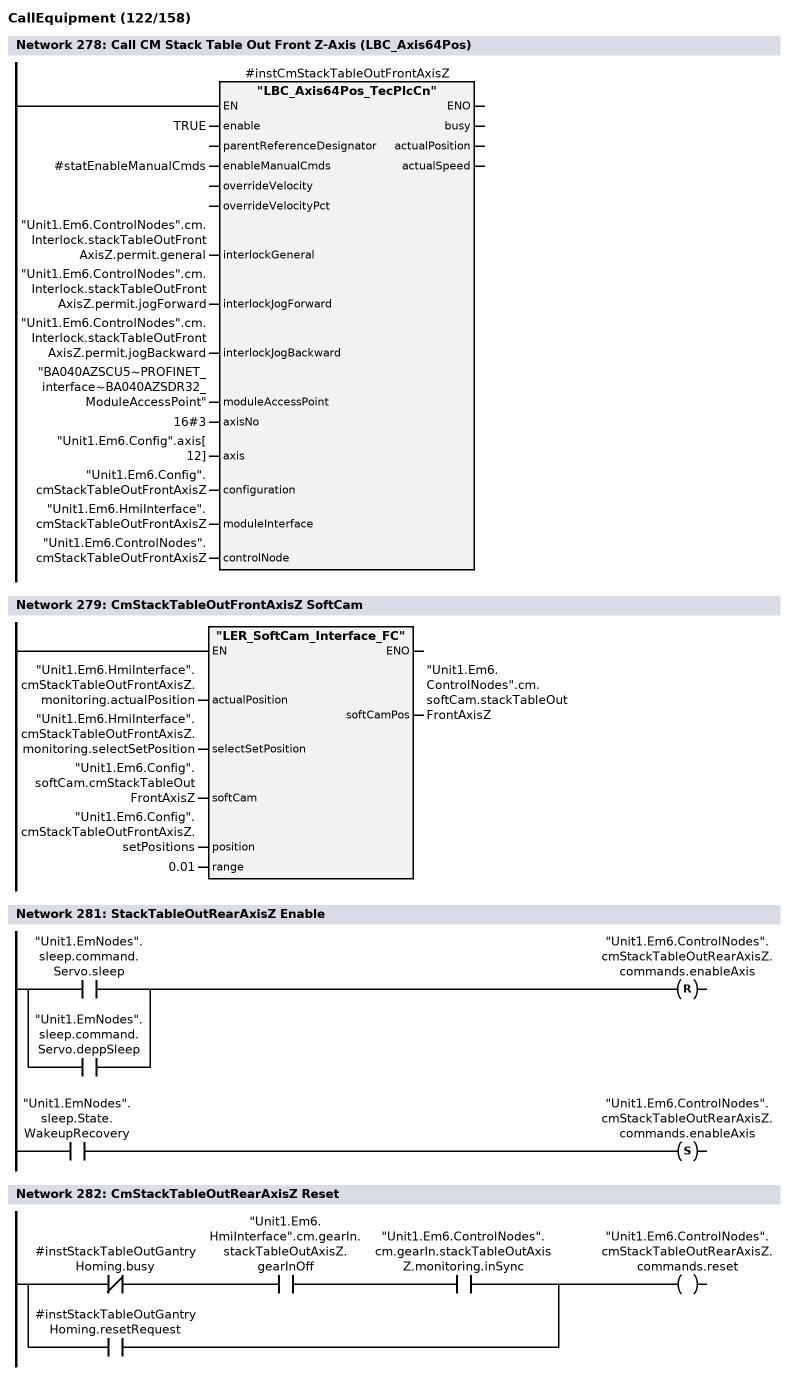
   RUNG wire#powerrail
      #instCmStackTableOutFrontAxisZ(enable := TRUE, parentReferenceDesignator :=, enableManualCmds := #statEnableManualCmds, overrideVelocity :=, overrideVelocityPct :=, interlockGeneral := "Unit1.Em6.ControlNodes".cm.Interlock.stackTableOutFrontAxisZ.permit.general, interlockJogForward := "Unit1.Em6.ControlNodes".cm.Interlock.stackTableOutFrontAxisZ.permit.jogForward, interlockJogBackward := "Unit1.Em6.ControlNodes".cm.Interlock.stackTableOutFrontAxisZ.permit.jogBackward, moduleAccessPoint := "BA040AZSCU5~PROFINET_interface~BA040AZSDR32_ModuleAccessPoint", axisNo := 16#3, axis := "Unit1.Em6.Config".axis[12], configuration := "Unit1.Em6.Config".cmStackTableOutFrontAxisZ, moduleInterface := "Unit1.Em6.HmiInterface".cmStackTableOutFrontAxisZ, controlNode := "Unit1.Em6.ControlNodes".cmStackTableOutFrontAxisZ, busy =>, actualPosition =>, actualSpeed =>)
   END_RUNG
   // the same network as SCL:
   #instCmStackTableOutFrontAxisZ(enable := TRUE,   // "LBC_Axis64Pos_TecPlcCn"
                           enableManualCmds := #statEnableManualCmds,
                           interlockGeneral := "Unit1.Em6.ControlNodes".cm.Interlock.stackTableOutFrontAxisZ.permit.general,
                           interlockJogForward := "Unit1.Em6.ControlNodes".cm.Interlock.stackTableOutFrontAxisZ.permit.jogForward,
                           interlockJogBackward := "Unit1.Em6.ControlNodes".cm.Interlock.stackTableOutFrontAxisZ.permit.jogBackward,
                           moduleAccessPoint := "BA040AZSCU5~PROFINET_interface~BA040AZSDR32_ModuleAccessPoint",
                           axisNo := 16#3,
                           axis := "Unit1.Em6.Config".axis[12],
                           configuration := "Unit1.Em6.Config".cmStackTableOutFrontAxisZ,
                           moduleInterface := "Unit1.Em6.HmiInterface".cmStackTableOutFrontAxisZ,
                           controlNode := "Unit1.Em6.ControlNodes".cmStackTableOutFrontAxisZ);
END_REGION

REGION Network 279: CmStackTableOutFrontAxisZ SoftCam
   RUNG wire#powerrail
      "LER_SoftCam_Interface_FC"(actualPosition := "Unit1.Em6.HmiInterface".cmStackTableOutFrontAxisZ.monitoring.actualPosition, selectSetPosition := "Unit1.Em6.HmiInterface".cmStackTableOutFrontAxisZ.monitoring.selectSetPosition, softCam := "Unit1.Em6.Config".softCam.cmStackTableOutFrontAxisZ, position := "Unit1.Em6.Config".cmStackTableOutFrontAxisZ.setPositions, range := 0.01, softCamPos => "Unit1.Em6.ControlNodes".cm.softCam.stackTableOutFrontAxisZ)
   END_RUNG
   // the same network as SCL:
   "LER_SoftCam_Interface_FC"(actualPosition := "Unit1.Em6.HmiInterface".cmStackTableOutFrontAxisZ.monitoring.actualPosition,
                           selectSetPosition := "Unit1.Em6.HmiInterface".cmStackTableOutFrontAxisZ.monitoring.selectSetPosition,
                           softCam := "Unit1.Em6.Config".softCam.cmStackTableOutFrontAxisZ,
                           position := "Unit1.Em6.Config".cmStackTableOutFrontAxisZ.setPositions,
                           range := 0.01,
                           softCamPos => "Unit1.Em6.ControlNodes".cm.softCam.stackTableOutFrontAxisZ);
END_REGION

REGION Network 281: StackTableOutRearAxisZ Enable
   RUNG wire#powerrail
      Contact( "Unit1.EmNodes".sleep.command.Servo.sleep )
      wire#w1
      R_Coil( "Unit1.Em6.ControlNodes".cmStackTableOutRearAxisZ.commands.enableAxis )
   END_RUNG
   RUNG wire#powerrail
      Contact( "Unit1.EmNodes".sleep.command.Servo.deppSleep )
   END_RUNG wire#w1
   RUNG wire#powerrail
      Contact( "Unit1.EmNodes".sleep.State.WakeupRecovery )
      S_Coil( "Unit1.Em6.ControlNodes".cmStackTableOutRearAxisZ.commands.enableAxis )
   END_RUNG
   // the same network as SCL:
   IF "Unit1.EmNodes".sleep.command.Servo.sleep OR "Unit1.EmNodes".sleep.command.Servo.deppSleep THEN
       "Unit1.Em6.ControlNodes".cmStackTableOutRearAxisZ.commands.enableAxis := FALSE;
   END_IF;
   IF "Unit1.EmNodes".sleep.State.WakeupRecovery THEN
       "Unit1.Em6.ControlNodes".cmStackTableOutRearAxisZ.commands.enableAxis := TRUE;
   END_IF;
END_REGION

REGION Network 282: CmStackTableOutRearAxisZ Reset
   RUNG wire#powerrail
      I_Contact( #instStackTableOutGantryHoming.busy )
      Contact( "Unit1.Em6.HmiInterface".cm.gearIn.stackTableOutAxisZ.gearInOff )
      Contact( "Unit1.Em6.ControlNodes".cm.gearIn.stackTableOutAxisZ.monitoring.inSync )
      wire#w1
      Coil( "Unit1.Em6.ControlNodes".cmStackTableOutRearAxisZ.commands.reset )
   END_RUNG
   RUNG wire#powerrail
      Contact( #instStackTableOutGantryHoming.resetRequest )
   END_RUNG wire#w1
   // the same network as SCL:
   "Unit1.Em6.ControlNodes".cmStackTableOutRearAxisZ.commands.reset := (NOT #instStackTableOutGantryHoming.busy AND "Unit1.Em6.HmiInterface".cm.gearIn.stackTableOutAxisZ.gearInOff AND "Unit1.Em6.ControlNodes".cm.gearIn.stackTableOutAxisZ.monitoring.inSync) OR #instStackTableOutGantryHoming.resetRequest;
END_REGION

REGION Network 283: CmStackTableOutRearAxisZ Home
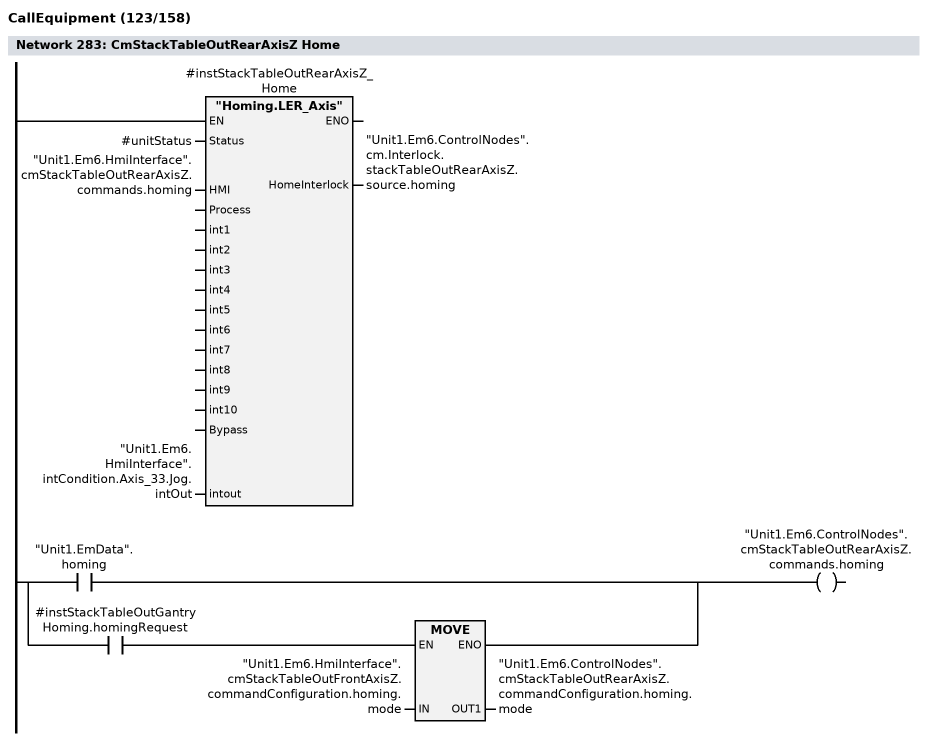
   RUNG wire#powerrail
      #instStackTableOutRearAxisZ_Home(Status := #unitStatus, HMI := "Unit1.Em6.HmiInterface".cmStackTableOutRearAxisZ.commands.homing, Process :=, int1 :=, int2 :=, int3 :=, int4 :=, int5 :=, int6 :=, int7 :=, int8 :=, int9 :=, int10 :=, Bypass :=, intout := "Unit1.Em6.HmiInterface".intCondition.Axis_33.Jog.intOut, HomeInterlock => "Unit1.Em6.ControlNodes".cm.Interlock.stackTableOutRearAxisZ.source.homing)
   END_RUNG
   RUNG wire#powerrail
      Contact( "Unit1.EmData".homing )
      wire#w1
      Coil( "Unit1.Em6.ControlNodes".cmStackTableOutRearAxisZ.commands.homing )
   END_RUNG
   RUNG wire#powerrail
      Contact( #instStackTableOutGantryHoming.homingRequest )
      Move(in := "Unit1.Em6.HmiInterface".cmStackTableOutFrontAxisZ.commandConfiguration.homing.mode, out1 => "Unit1.Em6.ControlNodes".cmStackTableOutRearAxisZ.commandConfiguration.homing.mode)
   END_RUNG wire#w1
   // the same network as SCL:
   #instStackTableOutRearAxisZ_Home(Status := #unitStatus,   // "Homing.LER_Axis"
                           HMI := "Unit1.Em6.HmiInterface".cmStackTableOutRearAxisZ.commands.homing,
                           intout := "Unit1.Em6.HmiInterface".intCondition.Axis_33.Jog.intOut,
                           HomeInterlock => "Unit1.Em6.ControlNodes".cm.Interlock.stackTableOutRearAxisZ.source.homing);
   IF #instStackTableOutGantryHoming.homingRequest THEN
       "Unit1.Em6.ControlNodes".cmStackTableOutRearAxisZ.commandConfiguration.homing.mode := "Unit1.Em6.HmiInterface".cmStackTableOutFrontAxisZ.commandConfiguration.homing.mode;
   END_IF;
   "Unit1.Em6.ControlNodes".cmStackTableOutRearAxisZ.commands.homing := "Unit1.EmData".homing OR #instStackTableOutGantryHoming.homingRequest;
END_REGION

REGION Network 284: CmStackTableOutRearAxisZ Position Absolute Jog
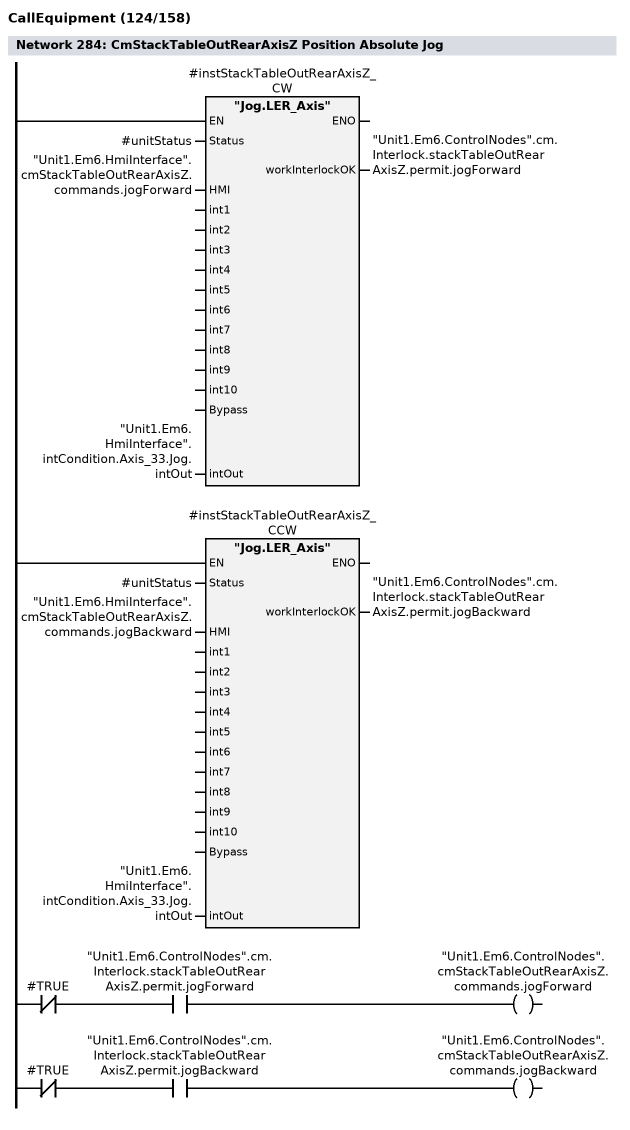
   RUNG wire#powerrail
      #instStackTableOutRearAxisZ_CW(Status := #unitStatus, HMI := "Unit1.Em6.HmiInterface".cmStackTableOutRearAxisZ.commands.jogForward, int1 :=, int2 :=, int3 :=, int4 :=, int5 :=, int6 :=, int7 :=, int8 :=, int9 :=, int10 :=, Bypass :=, intOut := "Unit1.Em6.HmiInterface".intCondition.Axis_33.Jog.intOut, workInterlockOK => "Unit1.Em6.ControlNodes".cm.Interlock.stackTableOutRearAxisZ.permit.jogForward)
   END_RUNG
   RUNG wire#powerrail
      #instStackTableOutRearAxisZ_CCW(Status := #unitStatus, HMI := "Unit1.Em6.HmiInterface".cmStackTableOutRearAxisZ.commands.jogBackward, int1 :=, int2 :=, int3 :=, int4 :=, int5 :=, int6 :=, int7 :=, int8 :=, int9 :=, int10 :=, Bypass :=, intOut := "Unit1.Em6.HmiInterface".intCondition.Axis_33.Jog.intOut, workInterlockOK => "Unit1.Em6.ControlNodes".cm.Interlock.stackTableOutRearAxisZ.permit.jogBackward)
   END_RUNG
   RUNG wire#powerrail
      I_Contact( #TRUE )
      Contact( "Unit1.Em6.ControlNodes".cm.Interlock.stackTableOutRearAxisZ.permit.jogForward )
      Coil( "Unit1.Em6.ControlNodes".cmStackTableOutRearAxisZ.commands.jogForward )
   END_RUNG
   RUNG wire#powerrail
      I_Contact( #TRUE )
      Contact( "Unit1.Em6.ControlNodes".cm.Interlock.stackTableOutRearAxisZ.permit.jogBackward )
      Coil( "Unit1.Em6.ControlNodes".cmStackTableOutRearAxisZ.commands.jogBackward )
   END_RUNG
   // the same network as SCL:
   #instStackTableOutRearAxisZ_CW(Status := #unitStatus,   // "Jog.LER_Axis"
                           HMI := "Unit1.Em6.HmiInterface".cmStackTableOutRearAxisZ.commands.jogForward,
                           intOut := "Unit1.Em6.HmiInterface".intCondition.Axis_33.Jog.intOut,
                           workInterlockOK => "Unit1.Em6.ControlNodes".cm.Interlock.stackTableOutRearAxisZ.permit.jogForward);
   #instStackTableOutRearAxisZ_CCW(Status := #unitStatus,   // "Jog.LER_Axis"
                           HMI := "Unit1.Em6.HmiInterface".cmStackTableOutRearAxisZ.commands.jogBackward,
                           intOut := "Unit1.Em6.HmiInterface".intCondition.Axis_33.Jog.intOut,
                           workInterlockOK => "Unit1.Em6.ControlNodes".cm.Interlock.stackTableOutRearAxisZ.permit.jogBackward);
   "Unit1.Em6.ControlNodes".cmStackTableOutRearAxisZ.commands.jogForward := NOT #TRUE AND "Unit1.Em6.ControlNodes".cm.Interlock.stackTableOutRearAxisZ.permit.jogForward;
   "Unit1.Em6.ControlNodes".cmStackTableOutRearAxisZ.commands.jogBackward := NOT #TRUE AND "Unit1.Em6.ControlNodes".cm.Interlock.stackTableOutRearAxisZ.permit.jogBackward;
END_REGION

REGION Network 285: CmStackTableOutRearAxisZ Position Absolute Position0
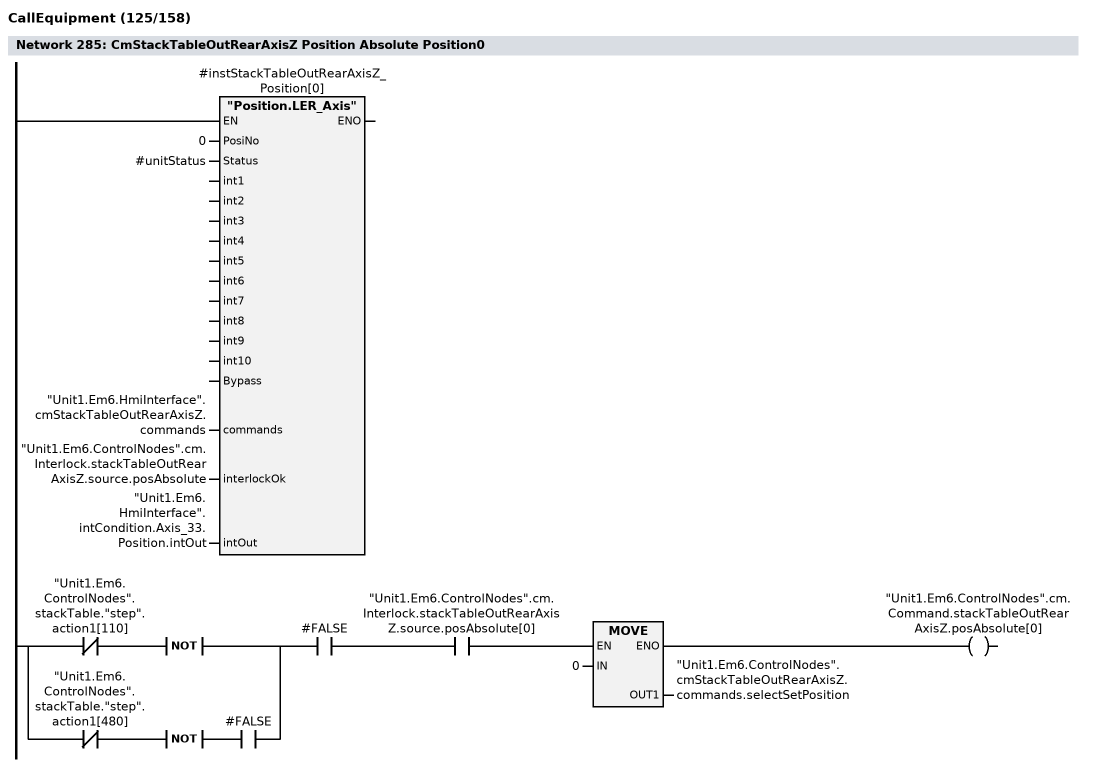
   RUNG wire#powerrail
      #instStackTableOutRearAxisZ_Position[0](PosiNo := 0, Status := #unitStatus, int1 :=, int2 :=, int3 :=, int4 :=, int5 :=, int6 :=, int7 :=, int8 :=, int9 :=, int10 :=, Bypass :=, commands := "Unit1.Em6.HmiInterface".cmStackTableOutRearAxisZ.commands, interlockOk := "Unit1.Em6.ControlNodes".cm.Interlock.stackTableOutRearAxisZ.source.posAbsolute, intOut := "Unit1.Em6.HmiInterface".intCondition.Axis_33.Position.intOut)
   END_RUNG
   RUNG wire#powerrail
      I_Contact( "Unit1.Em6.ControlNodes".stackTable."step".action1[110] )
      Not()
      wire#w1
      Contact( #FALSE )
      Contact( "Unit1.Em6.ControlNodes".cm.Interlock.stackTableOutRearAxisZ.source.posAbsolute[0] )
      Move(in := 0, out1 => "Unit1.Em6.ControlNodes".cmStackTableOutRearAxisZ.commands.selectSetPosition)
      Coil( "Unit1.Em6.ControlNodes".cm.Command.stackTableOutRearAxisZ.posAbsolute[0] )
   END_RUNG
   RUNG wire#powerrail
      I_Contact( "Unit1.Em6.ControlNodes".stackTable."step".action1[480] )
      Not()
      Contact( #FALSE )
   END_RUNG wire#w1
   // the same network as SCL:
   #instStackTableOutRearAxisZ_Position[0](PosiNo := 0,   // "Position.LER_Axis"
                           Status := #unitStatus,
                           commands := "Unit1.Em6.HmiInterface".cmStackTableOutRearAxisZ.commands,
                           interlockOk := "Unit1.Em6.ControlNodes".cm.Interlock.stackTableOutRearAxisZ.source.posAbsolute,
                           intOut := "Unit1.Em6.HmiInterface".intCondition.Axis_33.Position.intOut);
   #_w1 := (NOT (NOT "Unit1.Em6.ControlNodes".stackTable."step".action1[110]) OR (NOT (NOT "Unit1.Em6.ControlNodes".stackTable."step".action1[480]) AND #FALSE)) AND #FALSE AND "Unit1.Em6.ControlNodes".cm.Interlock.stackTableOutRearAxisZ.source.posAbsolute[0];
   IF #_w1 THEN "Unit1.Em6.ControlNodes".cmStackTableOutRearAxisZ.commands.selectSetPosition := 0; END_IF;
   "Unit1.Em6.ControlNodes".cm.Command.stackTableOutRearAxisZ.posAbsolute[0] := #_w1;
END_REGION

REGION Network 286: CmStackTableOutRearAxisZ Position Absolute Position1
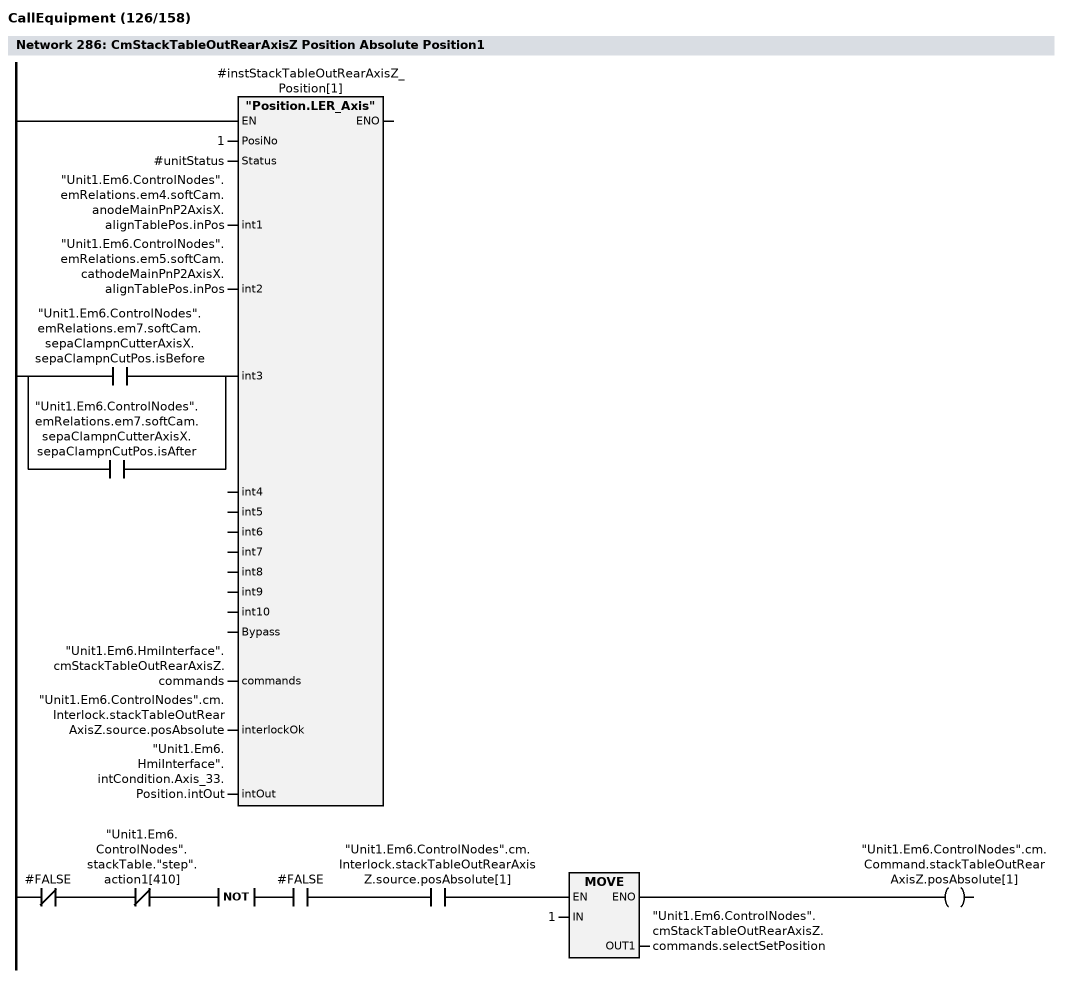
   RUNG wire#powerrail
      #instStackTableOutRearAxisZ_Position[1](int3 := wire#w1, PosiNo := 1, Status := #unitStatus, int1 := "Unit1.Em6.ControlNodes".emRelations.em4.softCam.anodeMainPnP2AxisX.alignTablePos.inPos, int2 := "Unit1.Em6.ControlNodes".emRelations.em5.softCam.cathodeMainPnP2AxisX.alignTablePos.inPos, int4 :=, int5 :=, int6 :=, int7 :=, int8 :=, int9 :=, int10 :=, Bypass :=, commands := "Unit1.Em6.HmiInterface".cmStackTableOutRearAxisZ.commands, interlockOk := "Unit1.Em6.ControlNodes".cm.Interlock.stackTableOutRearAxisZ.source.posAbsolute, intOut := "Unit1.Em6.HmiInterface".intCondition.Axis_33.Position.intOut)
   END_RUNG
   RUNG wire#powerrail
      Contact( "Unit1.Em6.ControlNodes".emRelations.em7.softCam.sepaClampnCutterAxisX.sepaClampnCutPos.isBefore )
   END_RUNG wire#w1
   RUNG wire#powerrail
      Contact( "Unit1.Em6.ControlNodes".emRelations.em7.softCam.sepaClampnCutterAxisX.sepaClampnCutPos.isAfter )
   END_RUNG wire#w1
   RUNG wire#powerrail
      I_Contact( #FALSE )
      I_Contact( "Unit1.Em6.ControlNodes".stackTable."step".action1[410] )
      Not()
      Contact( #FALSE )
      Contact( "Unit1.Em6.ControlNodes".cm.Interlock.stackTableOutRearAxisZ.source.posAbsolute[1] )
      Move(in := 1, out1 => "Unit1.Em6.ControlNodes".cmStackTableOutRearAxisZ.commands.selectSetPosition)
      Coil( "Unit1.Em6.ControlNodes".cm.Command.stackTableOutRearAxisZ.posAbsolute[1] )
   END_RUNG
   // the same network as SCL:
   #instStackTableOutRearAxisZ_Position[1](PosiNo := 1,   // "Position.LER_Axis"
                           Status := #unitStatus,
                           int1 := "Unit1.Em6.ControlNodes".emRelations.em4.softCam.anodeMainPnP2AxisX.alignTablePos.inPos,
                           int2 := "Unit1.Em6.ControlNodes".emRelations.em5.softCam.cathodeMainPnP2AxisX.alignTablePos.inPos,
                           int3 := "Unit1.Em6.ControlNodes".emRelations.em7.softCam.sepaClampnCutterAxisX.sepaClampnCutPos.isBefore OR "Unit1.Em6.ControlNodes".emRelations.em7.softCam.sepaClampnCutterAxisX.sepaClampnCutPos.isAfter,
                           commands := "Unit1.Em6.HmiInterface".cmStackTableOutRearAxisZ.commands,
                           interlockOk := "Unit1.Em6.ControlNodes".cm.Interlock.stackTableOutRearAxisZ.source.posAbsolute,
                           intOut := "Unit1.Em6.HmiInterface".intCondition.Axis_33.Position.intOut);
   #_w1 := NOT (NOT #FALSE AND NOT "Unit1.Em6.ControlNodes".stackTable."step".action1[410]) AND #FALSE AND "Unit1.Em6.ControlNodes".cm.Interlock.stackTableOutRearAxisZ.source.posAbsolute[1];
   IF #_w1 THEN "Unit1.Em6.ControlNodes".cmStackTableOutRearAxisZ.commands.selectSetPosition := 1; END_IF;
   "Unit1.Em6.ControlNodes".cm.Command.stackTableOutRearAxisZ.posAbsolute[1] := #_w1;
END_REGION

REGION Network 287: CmStackTableOutRearAxisZ Position Absolute Position2
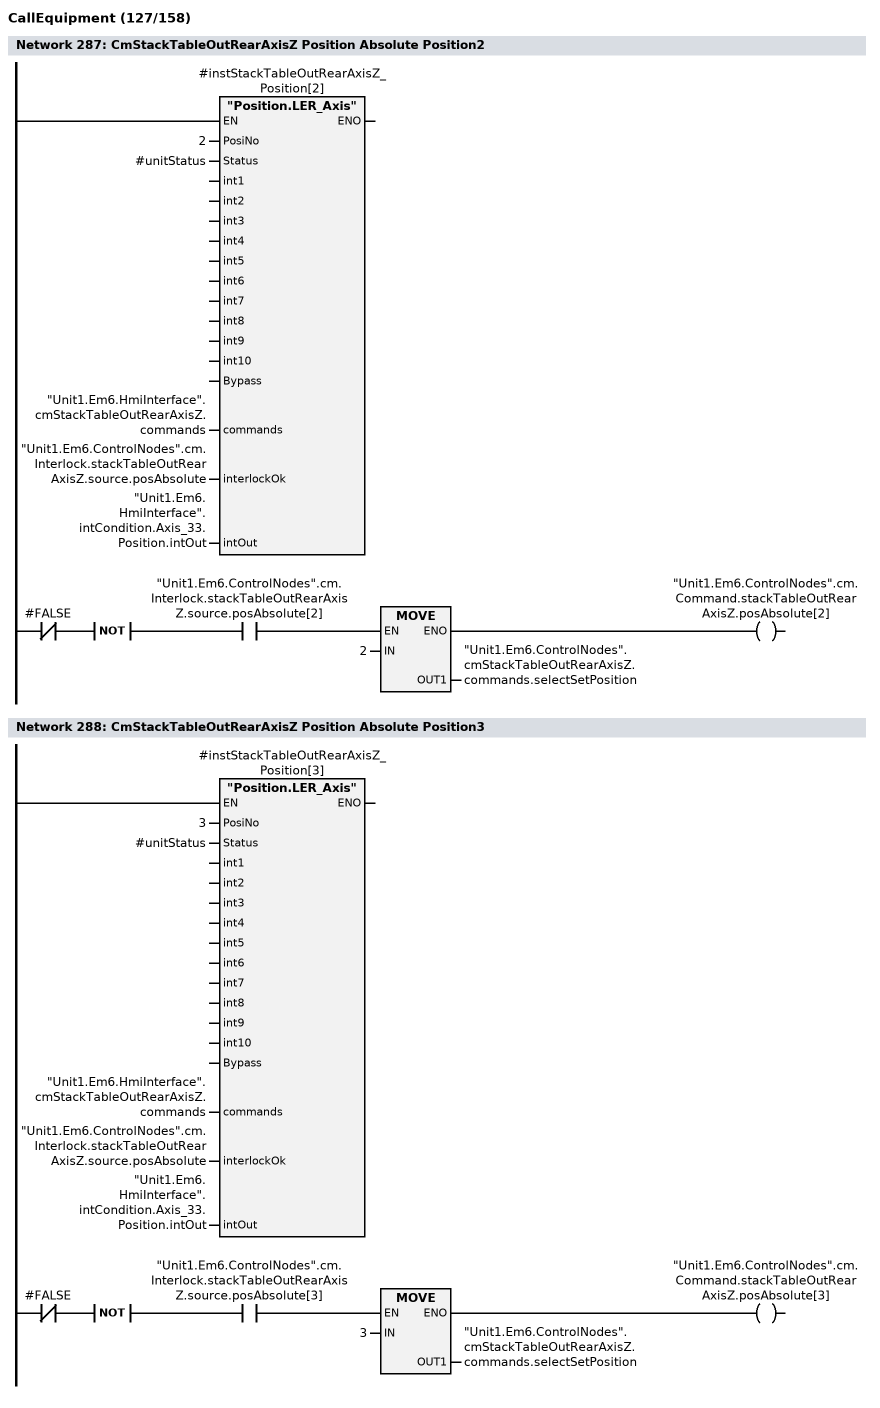
   RUNG wire#powerrail
      #instStackTableOutRearAxisZ_Position[2](PosiNo := 2, Status := #unitStatus, int1 :=, int2 :=, int3 :=, int4 :=, int5 :=, int6 :=, int7 :=, int8 :=, int9 :=, int10 :=, Bypass :=, commands := "Unit1.Em6.HmiInterface".cmStackTableOutRearAxisZ.commands, interlockOk := "Unit1.Em6.ControlNodes".cm.Interlock.stackTableOutRearAxisZ.source.posAbsolute, intOut := "Unit1.Em6.HmiInterface".intCondition.Axis_33.Position.intOut)
   END_RUNG
   RUNG wire#powerrail
      I_Contact( #FALSE )
      Not()
      Contact( "Unit1.Em6.ControlNodes".cm.Interlock.stackTableOutRearAxisZ.source.posAbsolute[2] )
      Move(in := 2, out1 => "Unit1.Em6.ControlNodes".cmStackTableOutRearAxisZ.commands.selectSetPosition)
      Coil( "Unit1.Em6.ControlNodes".cm.Command.stackTableOutRearAxisZ.posAbsolute[2] )
   END_RUNG
   // the same network as SCL:
   #instStackTableOutRearAxisZ_Position[2](PosiNo := 2,   // "Position.LER_Axis"
                           Status := #unitStatus,
                           commands := "Unit1.Em6.HmiInterface".cmStackTableOutRearAxisZ.commands,
                           interlockOk := "Unit1.Em6.ControlNodes".cm.Interlock.stackTableOutRearAxisZ.source.posAbsolute,
                           intOut := "Unit1.Em6.HmiInterface".intCondition.Axis_33.Position.intOut);
   #_w1 := NOT (NOT #FALSE) AND "Unit1.Em6.ControlNodes".cm.Interlock.stackTableOutRearAxisZ.source.posAbsolute[2];
   IF #_w1 THEN "Unit1.Em6.ControlNodes".cmStackTableOutRearAxisZ.commands.selectSetPosition := 2; END_IF;
   "Unit1.Em6.ControlNodes".cm.Command.stackTableOutRearAxisZ.posAbsolute[2] := #_w1;
END_REGION

REGION Network 288: CmStackTableOutRearAxisZ Position Absolute Position3
   RUNG wire#powerrail
      #instStackTableOutRearAxisZ_Position[3](PosiNo := 3, Status := #unitStatus, int1 :=, int2 :=, int3 :=, int4 :=, int5 :=, int6 :=, int7 :=, int8 :=, int9 :=, int10 :=, Bypass :=, commands := "Unit1.Em6.HmiInterface".cmStackTableOutRearAxisZ.commands, interlockOk := "Unit1.Em6.ControlNodes".cm.Interlock.stackTableOutRearAxisZ.source.posAbsolute, intOut := "Unit1.Em6.HmiInterface".intCondition.Axis_33.Position.intOut)
   END_RUNG
   RUNG wire#powerrail
      I_Contact( #FALSE )
      Not()
      Contact( "Unit1.Em6.ControlNodes".cm.Interlock.stackTableOutRearAxisZ.source.posAbsolute[3] )
      Move(in := 3, out1 => "Unit1.Em6.ControlNodes".cmStackTableOutRearAxisZ.commands.selectSetPosition)
      Coil( "Unit1.Em6.ControlNodes".cm.Command.stackTableOutRearAxisZ.posAbsolute[3] )
   END_RUNG
   // the same network as SCL:
   #instStackTableOutRearAxisZ_Position[3](PosiNo := 3,   // "Position.LER_Axis"
                           Status := #unitStatus,
                           commands := "Unit1.Em6.HmiInterface".cmStackTableOutRearAxisZ.commands,
                           interlockOk := "Unit1.Em6.ControlNodes".cm.Interlock.stackTableOutRearAxisZ.source.posAbsolute,
                           intOut := "Unit1.Em6.HmiInterface".intCondition.Axis_33.Position.intOut);
   #_w1 := NOT (NOT #FALSE) AND "Unit1.Em6.ControlNodes".cm.Interlock.stackTableOutRearAxisZ.source.posAbsolute[3];
   IF #_w1 THEN "Unit1.Em6.ControlNodes".cmStackTableOutRearAxisZ.commands.selectSetPosition := 3; END_IF;
   "Unit1.Em6.ControlNodes".cm.Command.stackTableOutRearAxisZ.posAbsolute[3] := #_w1;
END_REGION

REGION Network 289: CmStackTableOutRearAxisZ Position Absolute Position4
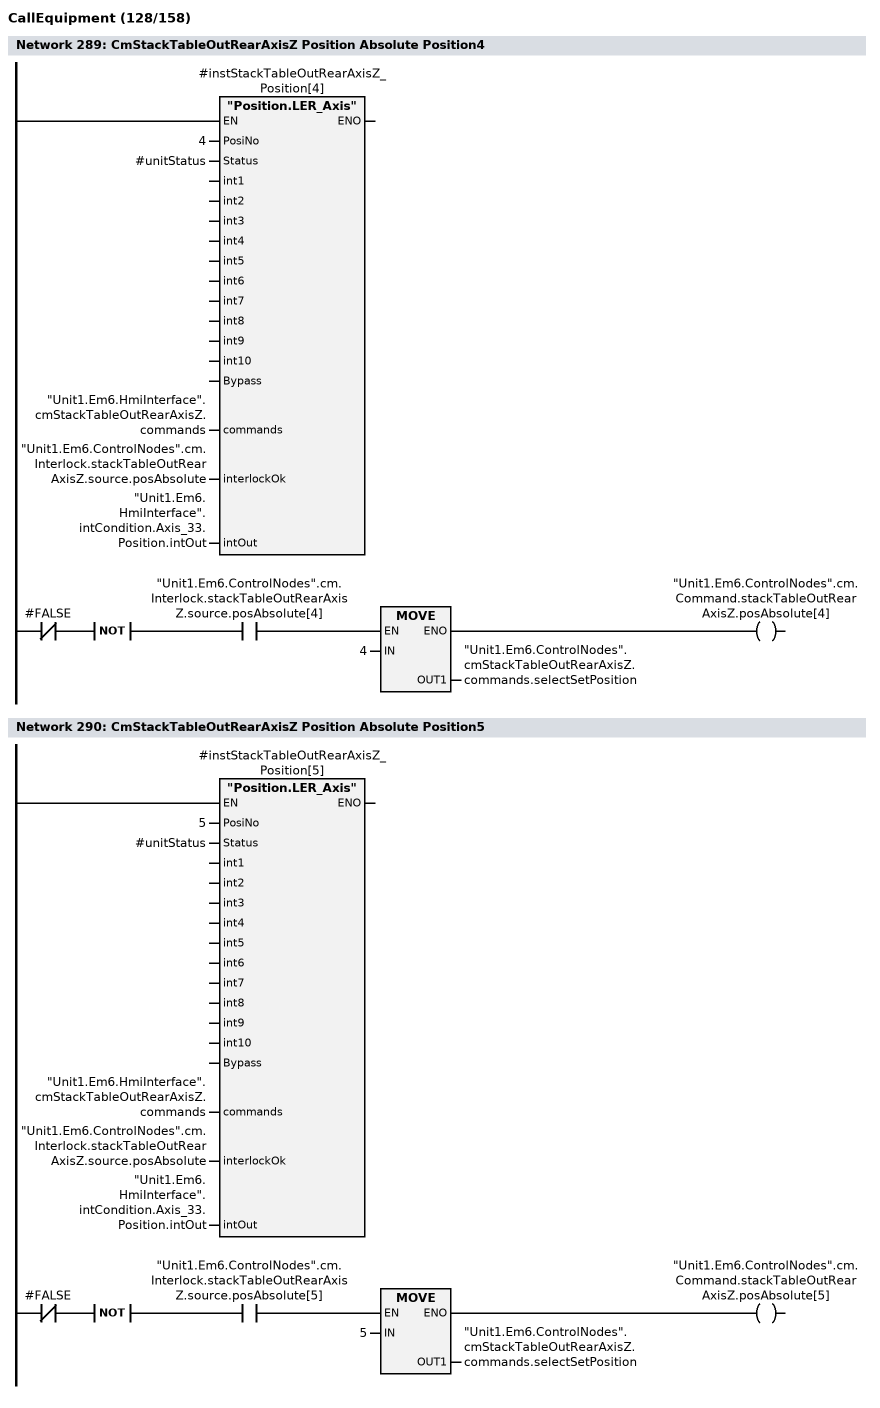
   RUNG wire#powerrail
      #instStackTableOutRearAxisZ_Position[4](PosiNo := 4, Status := #unitStatus, int1 :=, int2 :=, int3 :=, int4 :=, int5 :=, int6 :=, int7 :=, int8 :=, int9 :=, int10 :=, Bypass :=, commands := "Unit1.Em6.HmiInterface".cmStackTableOutRearAxisZ.commands, interlockOk := "Unit1.Em6.ControlNodes".cm.Interlock.stackTableOutRearAxisZ.source.posAbsolute, intOut := "Unit1.Em6.HmiInterface".intCondition.Axis_33.Position.intOut)
   END_RUNG
   RUNG wire#powerrail
      I_Contact( #FALSE )
      Not()
      Contact( "Unit1.Em6.ControlNodes".cm.Interlock.stackTableOutRearAxisZ.source.posAbsolute[4] )
      Move(in := 4, out1 => "Unit1.Em6.ControlNodes".cmStackTableOutRearAxisZ.commands.selectSetPosition)
      Coil( "Unit1.Em6.ControlNodes".cm.Command.stackTableOutRearAxisZ.posAbsolute[4] )
   END_RUNG
   // the same network as SCL:
   #instStackTableOutRearAxisZ_Position[4](PosiNo := 4,   // "Position.LER_Axis"
                           Status := #unitStatus,
                           commands := "Unit1.Em6.HmiInterface".cmStackTableOutRearAxisZ.commands,
                           interlockOk := "Unit1.Em6.ControlNodes".cm.Interlock.stackTableOutRearAxisZ.source.posAbsolute,
                           intOut := "Unit1.Em6.HmiInterface".intCondition.Axis_33.Position.intOut);
   #_w1 := NOT (NOT #FALSE) AND "Unit1.Em6.ControlNodes".cm.Interlock.stackTableOutRearAxisZ.source.posAbsolute[4];
   IF #_w1 THEN "Unit1.Em6.ControlNodes".cmStackTableOutRearAxisZ.commands.selectSetPosition := 4; END_IF;
   "Unit1.Em6.ControlNodes".cm.Command.stackTableOutRearAxisZ.posAbsolute[4] := #_w1;
END_REGION

REGION Network 290: CmStackTableOutRearAxisZ Position Absolute Position5
   RUNG wire#powerrail
      #instStackTableOutRearAxisZ_Position[5](PosiNo := 5, Status := #unitStatus, int1 :=, int2 :=, int3 :=, int4 :=, int5 :=, int6 :=, int7 :=, int8 :=, int9 :=, int10 :=, Bypass :=, commands := "Unit1.Em6.HmiInterface".cmStackTableOutRearAxisZ.commands, interlockOk := "Unit1.Em6.ControlNodes".cm.Interlock.stackTableOutRearAxisZ.source.posAbsolute, intOut := "Unit1.Em6.HmiInterface".intCondition.Axis_33.Position.intOut)
   END_RUNG
   RUNG wire#powerrail
      I_Contact( #FALSE )
      Not()
      Contact( "Unit1.Em6.ControlNodes".cm.Interlock.stackTableOutRearAxisZ.source.posAbsolute[5] )
      Move(in := 5, out1 => "Unit1.Em6.ControlNodes".cmStackTableOutRearAxisZ.commands.selectSetPosition)
      Coil( "Unit1.Em6.ControlNodes".cm.Command.stackTableOutRearAxisZ.posAbsolute[5] )
   END_RUNG
   // the same network as SCL:
   #instStackTableOutRearAxisZ_Position[5](PosiNo := 5,   // "Position.LER_Axis"
                           Status := #unitStatus,
                           commands := "Unit1.Em6.HmiInterface".cmStackTableOutRearAxisZ.commands,
                           interlockOk := "Unit1.Em6.ControlNodes".cm.Interlock.stackTableOutRearAxisZ.source.posAbsolute,
                           intOut := "Unit1.Em6.HmiInterface".intCondition.Axis_33.Position.intOut);
   #_w1 := NOT (NOT #FALSE) AND "Unit1.Em6.ControlNodes".cm.Interlock.stackTableOutRearAxisZ.source.posAbsolute[5];
   IF #_w1 THEN "Unit1.Em6.ControlNodes".cmStackTableOutRearAxisZ.commands.selectSetPosition := 5; END_IF;
   "Unit1.Em6.ControlNodes".cm.Command.stackTableOutRearAxisZ.posAbsolute[5] := #_w1;
END_REGION

REGION Network 291: CmStackTableOutRearAxisZ Summary Command
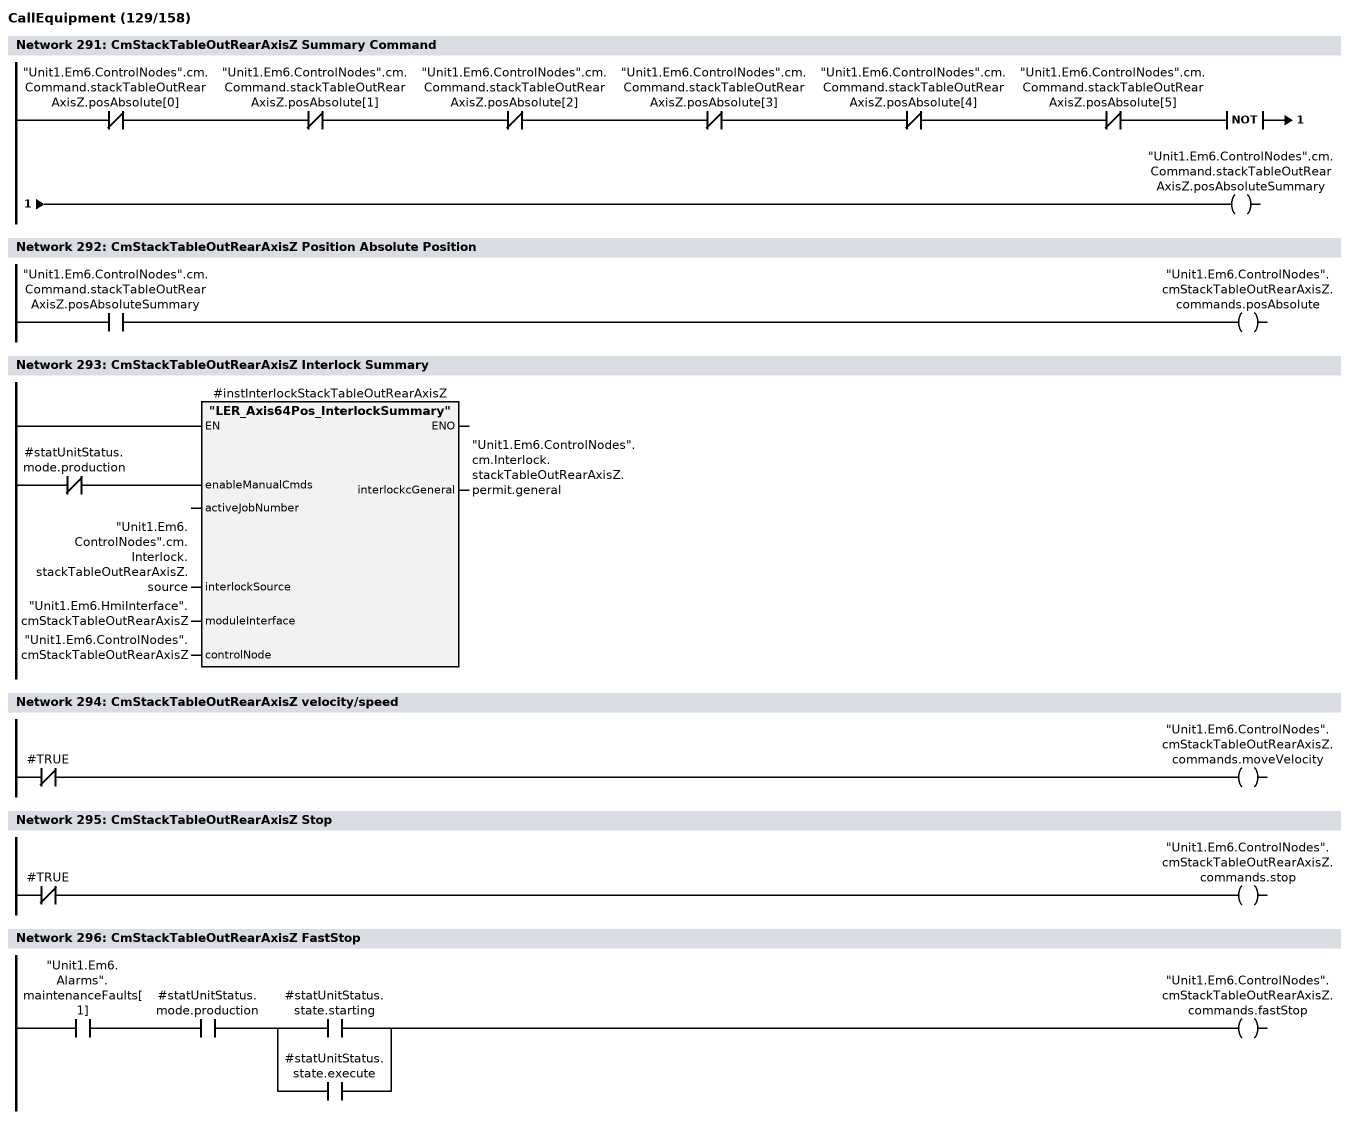
   RUNG wire#powerrail
      I_Contact( "Unit1.Em6.ControlNodes".cm.Command.stackTableOutRearAxisZ.posAbsolute[0] )
      I_Contact( "Unit1.Em6.ControlNodes".cm.Command.stackTableOutRearAxisZ.posAbsolute[1] )
      I_Contact( "Unit1.Em6.ControlNodes".cm.Command.stackTableOutRearAxisZ.posAbsolute[2] )
      I_Contact( "Unit1.Em6.ControlNodes".cm.Command.stackTableOutRearAxisZ.posAbsolute[3] )
      I_Contact( "Unit1.Em6.ControlNodes".cm.Command.stackTableOutRearAxisZ.posAbsolute[4] )
      I_Contact( "Unit1.Em6.ControlNodes".cm.Command.stackTableOutRearAxisZ.posAbsolute[5] )
      Not()
      Coil( "Unit1.Em6.ControlNodes".cm.Command.stackTableOutRearAxisZ.posAbsoluteSummary )
   END_RUNG
   // the same network as SCL:
   "Unit1.Em6.ControlNodes".cm.Command.stackTableOutRearAxisZ.posAbsoluteSummary := NOT (NOT "Unit1.Em6.ControlNodes".cm.Command.stackTableOutRearAxisZ.posAbsolute[0] AND NOT "Unit1.Em6.ControlNodes".cm.Command.stackTableOutRearAxisZ.posAbsolute[1] AND NOT "Unit1.Em6.ControlNodes".cm.Command.stackTableOutRearAxisZ.posAbsolute[2] AND NOT "Unit1.Em6.ControlNodes".cm.Command.stackTableOutRearAxisZ.posAbsolute[3] AND NOT "Unit1.Em6.ControlNodes".cm.Command.stackTableOutRearAxisZ.posAbsolute[4] AND NOT "Unit1.Em6.ControlNodes".cm.Command.stackTableOutRearAxisZ.posAbsolute[5]);
END_REGION

REGION Network 292: CmStackTableOutRearAxisZ Position Absolute Position
   RUNG wire#powerrail
      Contact( "Unit1.Em6.ControlNodes".cm.Command.stackTableOutRearAxisZ.posAbsoluteSummary )
      Coil( "Unit1.Em6.ControlNodes".cmStackTableOutRearAxisZ.commands.posAbsolute )
   END_RUNG
   // the same network as SCL:
   "Unit1.Em6.ControlNodes".cmStackTableOutRearAxisZ.commands.posAbsolute := "Unit1.Em6.ControlNodes".cm.Command.stackTableOutRearAxisZ.posAbsoluteSummary;
END_REGION

REGION Network 293: CmStackTableOutRearAxisZ Interlock Summary
   RUNG wire#powerrail
      #instInterlockStackTableOutRearAxisZ(enableManualCmds := wire#w1, activeJobNumber :=, interlockSource := "Unit1.Em6.ControlNodes".cm.Interlock.stackTableOutRearAxisZ.source, moduleInterface := "Unit1.Em6.HmiInterface".cmStackTableOutRearAxisZ, controlNode := "Unit1.Em6.ControlNodes".cmStackTableOutRearAxisZ, interlockcGeneral => "Unit1.Em6.ControlNodes".cm.Interlock.stackTableOutRearAxisZ.permit.general)
   END_RUNG
   RUNG wire#powerrail
      I_Contact( #statUnitStatus.mode.production )
   END_RUNG wire#w1
   // the same network as SCL:
   #instInterlockStackTableOutRearAxisZ(enableManualCmds := NOT #statUnitStatus.mode.production,   // "LER_Axis64Pos_InterlockSummary"
                           interlockSource := "Unit1.Em6.ControlNodes".cm.Interlock.stackTableOutRearAxisZ.source,
                           moduleInterface := "Unit1.Em6.HmiInterface".cmStackTableOutRearAxisZ,
                           controlNode := "Unit1.Em6.ControlNodes".cmStackTableOutRearAxisZ,
                           interlockcGeneral => "Unit1.Em6.ControlNodes".cm.Interlock.stackTableOutRearAxisZ.permit.general);
END_REGION

REGION Network 294: CmStackTableOutRearAxisZ velocity/speed
   RUNG wire#powerrail
      I_Contact( #TRUE )
      Coil( "Unit1.Em6.ControlNodes".cmStackTableOutRearAxisZ.commands.moveVelocity )
   END_RUNG
   // the same network as SCL:
   "Unit1.Em6.ControlNodes".cmStackTableOutRearAxisZ.commands.moveVelocity := NOT #TRUE;
END_REGION

REGION Network 295: CmStackTableOutRearAxisZ Stop
   RUNG wire#powerrail
      I_Contact( #TRUE )
      Coil( "Unit1.Em6.ControlNodes".cmStackTableOutRearAxisZ.commands.stop )
   END_RUNG
   // the same network as SCL:
   "Unit1.Em6.ControlNodes".cmStackTableOutRearAxisZ.commands.stop := NOT #TRUE;
END_REGION

REGION Network 296: CmStackTableOutRearAxisZ FastStop
   RUNG wire#powerrail
      Contact( "Unit1.Em6.Alarms".maintenanceFaults[1] )
      Contact( #statUnitStatus.mode.production )
      wire#w1
      Contact( #statUnitStatus.state.starting )
      wire#w2
      Coil( "Unit1.Em6.ControlNodes".cmStackTableOutRearAxisZ.commands.fastStop )
   END_RUNG
   RUNG wire#w1
      Contact( #statUnitStatus.state.execute )
   END_RUNG wire#w2
   // the same network as SCL:
   "Unit1.Em6.ControlNodes".cmStackTableOutRearAxisZ.commands.fastStop := "Unit1.Em6.Alarms".maintenanceFaults[1] AND #statUnitStatus.mode.production AND (#statUnitStatus.state.starting OR #statUnitStatus.state.execute);
END_REGION

REGION Network 297: Call CM Stack Table Out Rear Z-Axis (LBC_Axis64Pos)
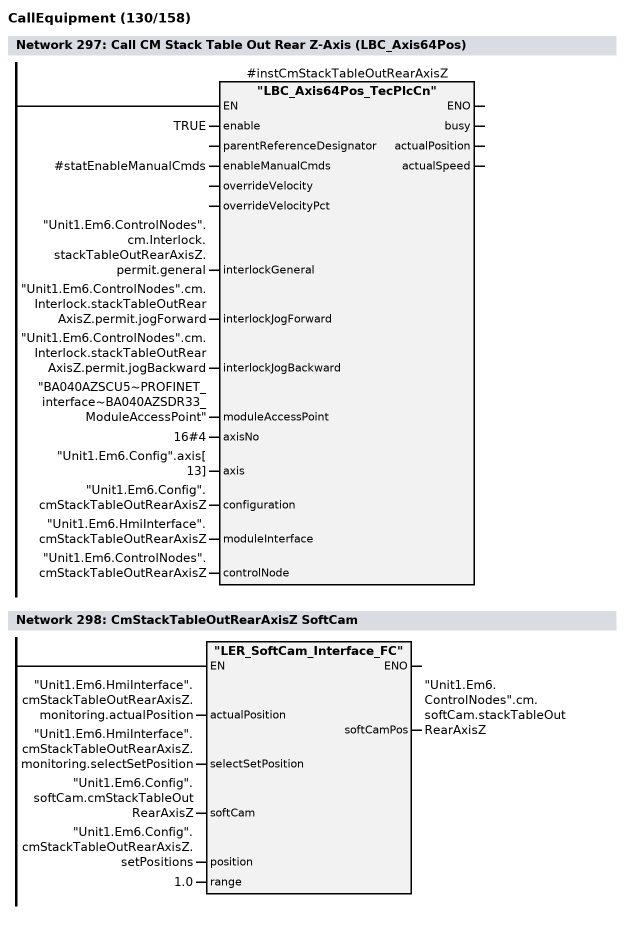
   RUNG wire#powerrail
      #instCmStackTableOutRearAxisZ(enable := TRUE, parentReferenceDesignator :=, enableManualCmds := #statEnableManualCmds, overrideVelocity :=, overrideVelocityPct :=, interlockGeneral := "Unit1.Em6.ControlNodes".cm.Interlock.stackTableOutRearAxisZ.permit.general, interlockJogForward := "Unit1.Em6.ControlNodes".cm.Interlock.stackTableOutRearAxisZ.permit.jogForward, interlockJogBackward := "Unit1.Em6.ControlNodes".cm.Interlock.stackTableOutRearAxisZ.permit.jogBackward, moduleAccessPoint := "BA040AZSCU5~PROFINET_interface~BA040AZSDR33_ModuleAccessPoint", axisNo := 16#4, axis := "Unit1.Em6.Config".axis[13], configuration := "Unit1.Em6.Config".cmStackTableOutRearAxisZ, moduleInterface := "Unit1.Em6.HmiInterface".cmStackTableOutRearAxisZ, controlNode := "Unit1.Em6.ControlNodes".cmStackTableOutRearAxisZ, busy =>, actualPosition =>, actualSpeed =>)
   END_RUNG
   // the same network as SCL:
   #instCmStackTableOutRearAxisZ(enable := TRUE,   // "LBC_Axis64Pos_TecPlcCn"
                           enableManualCmds := #statEnableManualCmds,
                           interlockGeneral := "Unit1.Em6.ControlNodes".cm.Interlock.stackTableOutRearAxisZ.permit.general,
                           interlockJogForward := "Unit1.Em6.ControlNodes".cm.Interlock.stackTableOutRearAxisZ.permit.jogForward,
                           interlockJogBackward := "Unit1.Em6.ControlNodes".cm.Interlock.stackTableOutRearAxisZ.permit.jogBackward,
                           moduleAccessPoint := "BA040AZSCU5~PROFINET_interface~BA040AZSDR33_ModuleAccessPoint",
                           axisNo := 16#4,
                           axis := "Unit1.Em6.Config".axis[13],
                           configuration := "Unit1.Em6.Config".cmStackTableOutRearAxisZ,
                           moduleInterface := "Unit1.Em6.HmiInterface".cmStackTableOutRearAxisZ,
                           controlNode := "Unit1.Em6.ControlNodes".cmStackTableOutRearAxisZ);
END_REGION

REGION Network 298: CmStackTableOutRearAxisZ SoftCam
   RUNG wire#powerrail
      "LER_SoftCam_Interface_FC"(actualPosition := "Unit1.Em6.HmiInterface".cmStackTableOutRearAxisZ.monitoring.actualPosition, selectSetPosition := "Unit1.Em6.HmiInterface".cmStackTableOutRearAxisZ.monitoring.selectSetPosition, softCam := "Unit1.Em6.Config".softCam.cmStackTableOutRearAxisZ, position := "Unit1.Em6.Config".cmStackTableOutRearAxisZ.setPositions, range := 1.0, softCamPos => "Unit1.Em6.ControlNodes".cm.softCam.stackTableOutRearAxisZ)
   END_RUNG
   // the same network as SCL:
   "LER_SoftCam_Interface_FC"(actualPosition := "Unit1.Em6.HmiInterface".cmStackTableOutRearAxisZ.monitoring.actualPosition,
                           selectSetPosition := "Unit1.Em6.HmiInterface".cmStackTableOutRearAxisZ.monitoring.selectSetPosition,
                           softCam := "Unit1.Em6.Config".softCam.cmStackTableOutRearAxisZ,
                           position := "Unit1.Em6.Config".cmStackTableOutRearAxisZ.setPositions,
                           range := 1.0,
                           softCamPos => "Unit1.Em6.ControlNodes".cm.softCam.stackTableOutRearAxisZ);
END_REGION

REGION Network 299: ******************** Brake Test (Axis) ********************
END_REGION

REGION Network 300: Mendrel Anode Front Z-Axis Brake Test
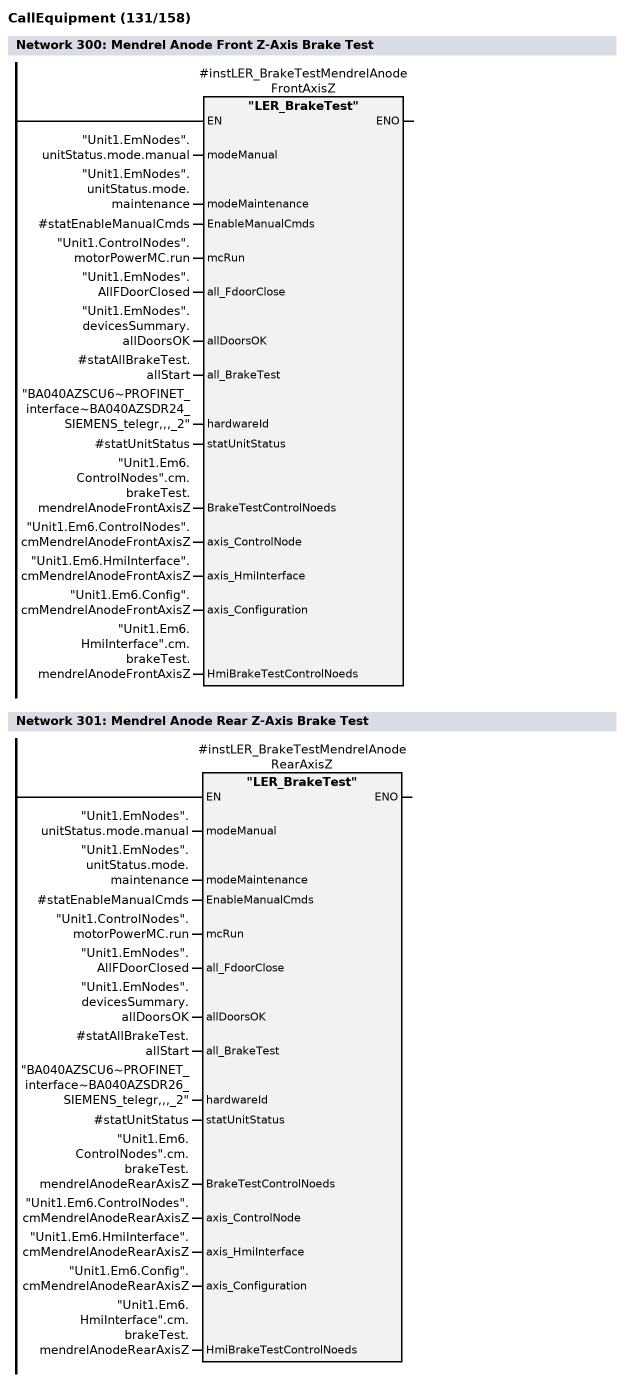
   RUNG wire#powerrail
      #instLER_BrakeTestMendrelAnodeFrontAxisZ(modeManual := "Unit1.EmNodes".unitStatus.mode.manual, modeMaintenance := "Unit1.EmNodes".unitStatus.mode.maintenance, EnableManualCmds := #statEnableManualCmds, mcRun := "Unit1.ControlNodes".motorPowerMC.run, all_FdoorClose := "Unit1.EmNodes".AllFDoorClosed, allDoorsOK := "Unit1.EmNodes".devicesSummary.allDoorsOK, all_BrakeTest := #statAllBrakeTest.allStart, hardwareId := "BA040AZSCU6~PROFINET_interface~BA040AZSDR24_SIEMENS_telegr,,,_2", statUnitStatus := #statUnitStatus, BrakeTestControlNoeds := "Unit1.Em6.ControlNodes".cm.brakeTest.mendrelAnodeFrontAxisZ, axis_ControlNode := "Unit1.Em6.ControlNodes".cmMendrelAnodeFrontAxisZ, axis_HmiInterface := "Unit1.Em6.HmiInterface".cmMendrelAnodeFrontAxisZ, axis_Configuration := "Unit1.Em6.Config".cmMendrelAnodeFrontAxisZ, HmiBrakeTestControlNoeds := "Unit1.Em6.HmiInterface".cm.brakeTest.mendrelAnodeFrontAxisZ)
   END_RUNG
   // the same network as SCL:
   #instLER_BrakeTestMendrelAnodeFrontAxisZ(modeManual := "Unit1.EmNodes".unitStatus.mode.manual,   // "LER_BrakeTest"
                           modeMaintenance := "Unit1.EmNodes".unitStatus.mode.maintenance,
                           EnableManualCmds := #statEnableManualCmds,
                           mcRun := "Unit1.ControlNodes".motorPowerMC.run,
                           all_FdoorClose := "Unit1.EmNodes".AllFDoorClosed,
                           allDoorsOK := "Unit1.EmNodes".devicesSummary.allDoorsOK,
                           all_BrakeTest := #statAllBrakeTest.allStart,
                           hardwareId := "BA040AZSCU6~PROFINET_interface~BA040AZSDR24_SIEMENS_telegr,,,_2",
                           statUnitStatus := #statUnitStatus,
                           BrakeTestControlNoeds := "Unit1.Em6.ControlNodes".cm.brakeTest.mendrelAnodeFrontAxisZ,
                           axis_ControlNode := "Unit1.Em6.ControlNodes".cmMendrelAnodeFrontAxisZ,
                           axis_HmiInterface := "Unit1.Em6.HmiInterface".cmMendrelAnodeFrontAxisZ,
                           axis_Configuration := "Unit1.Em6.Config".cmMendrelAnodeFrontAxisZ,
                           HmiBrakeTestControlNoeds := "Unit1.Em6.HmiInterface".cm.brakeTest.mendrelAnodeFrontAxisZ);
END_REGION

REGION Network 301: Mendrel Anode Rear Z-Axis Brake Test
   RUNG wire#powerrail
      #instLER_BrakeTestMendrelAnodeRearAxisZ(modeManual := "Unit1.EmNodes".unitStatus.mode.manual, modeMaintenance := "Unit1.EmNodes".unitStatus.mode.maintenance, EnableManualCmds := #statEnableManualCmds, mcRun := "Unit1.ControlNodes".motorPowerMC.run, all_FdoorClose := "Unit1.EmNodes".AllFDoorClosed, allDoorsOK := "Unit1.EmNodes".devicesSummary.allDoorsOK, all_BrakeTest := #statAllBrakeTest.allStart, hardwareId := "BA040AZSCU6~PROFINET_interface~BA040AZSDR26_SIEMENS_telegr,,,_2", statUnitStatus := #statUnitStatus, BrakeTestControlNoeds := "Unit1.Em6.ControlNodes".cm.brakeTest.mendrelAnodeRearAxisZ, axis_ControlNode := "Unit1.Em6.ControlNodes".cmMendrelAnodeRearAxisZ, axis_HmiInterface := "Unit1.Em6.HmiInterface".cmMendrelAnodeRearAxisZ, axis_Configuration := "Unit1.Em6.Config".cmMendrelAnodeRearAxisZ, HmiBrakeTestControlNoeds := "Unit1.Em6.HmiInterface".cm.brakeTest.mendrelAnodeRearAxisZ)
   END_RUNG
   // the same network as SCL:
   #instLER_BrakeTestMendrelAnodeRearAxisZ(modeManual := "Unit1.EmNodes".unitStatus.mode.manual,   // "LER_BrakeTest"
                           modeMaintenance := "Unit1.EmNodes".unitStatus.mode.maintenance,
                           EnableManualCmds := #statEnableManualCmds,
                           mcRun := "Unit1.ControlNodes".motorPowerMC.run,
                           all_FdoorClose := "Unit1.EmNodes".AllFDoorClosed,
                           allDoorsOK := "Unit1.EmNodes".devicesSummary.allDoorsOK,
                           all_BrakeTest := #statAllBrakeTest.allStart,
                           hardwareId := "BA040AZSCU6~PROFINET_interface~BA040AZSDR26_SIEMENS_telegr,,,_2",
                           statUnitStatus := #statUnitStatus,
                           BrakeTestControlNoeds := "Unit1.Em6.ControlNodes".cm.brakeTest.mendrelAnodeRearAxisZ,
                           axis_ControlNode := "Unit1.Em6.ControlNodes".cmMendrelAnodeRearAxisZ,
                           axis_HmiInterface := "Unit1.Em6.HmiInterface".cmMendrelAnodeRearAxisZ,
                           axis_Configuration := "Unit1.Em6.Config".cmMendrelAnodeRearAxisZ,
                           HmiBrakeTestControlNoeds := "Unit1.Em6.HmiInterface".cm.brakeTest.mendrelAnodeRearAxisZ);
END_REGION

REGION Network 302: Mendrel Cathode Front Z-Axis Brake Test
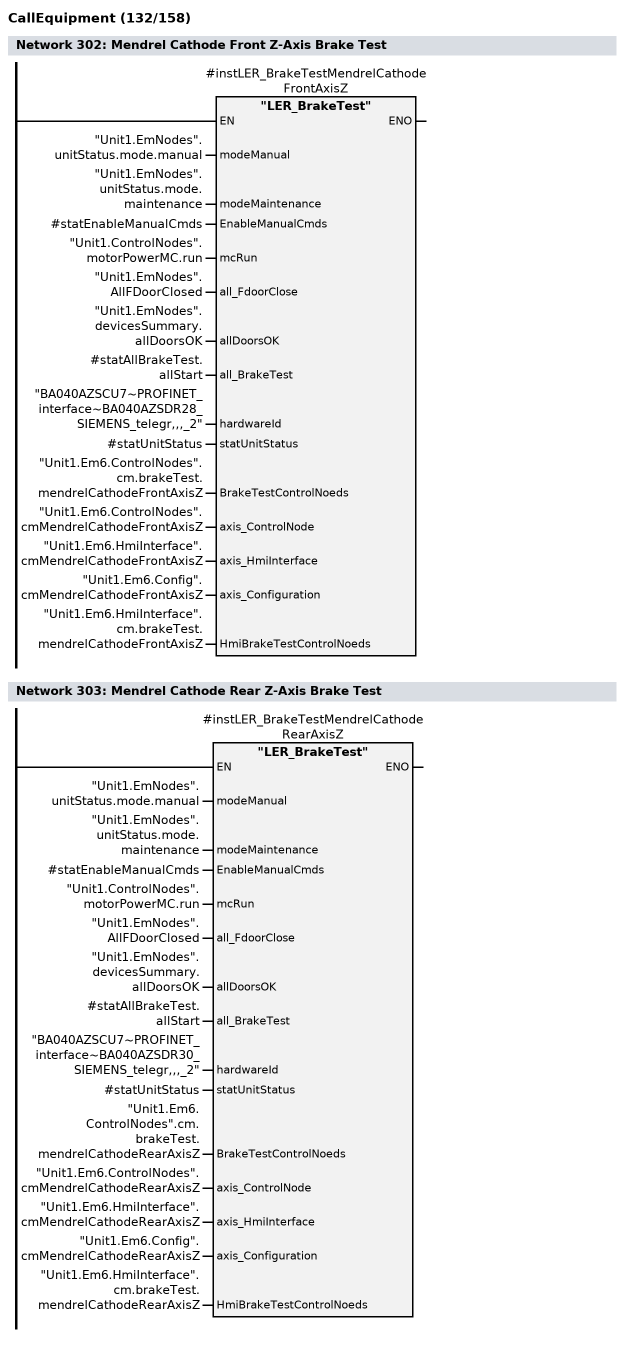
   RUNG wire#powerrail
      #instLER_BrakeTestMendrelCathodeFrontAxisZ(modeManual := "Unit1.EmNodes".unitStatus.mode.manual, modeMaintenance := "Unit1.EmNodes".unitStatus.mode.maintenance, EnableManualCmds := #statEnableManualCmds, mcRun := "Unit1.ControlNodes".motorPowerMC.run, all_FdoorClose := "Unit1.EmNodes".AllFDoorClosed, allDoorsOK := "Unit1.EmNodes".devicesSummary.allDoorsOK, all_BrakeTest := #statAllBrakeTest.allStart, hardwareId := "BA040AZSCU7~PROFINET_interface~BA040AZSDR28_SIEMENS_telegr,,,_2", statUnitStatus := #statUnitStatus, BrakeTestControlNoeds := "Unit1.Em6.ControlNodes".cm.brakeTest.mendrelCathodeFrontAxisZ, axis_ControlNode := "Unit1.Em6.ControlNodes".cmMendrelCathodeFrontAxisZ, axis_HmiInterface := "Unit1.Em6.HmiInterface".cmMendrelCathodeFrontAxisZ, axis_Configuration := "Unit1.Em6.Config".cmMendrelCathodeFrontAxisZ, HmiBrakeTestControlNoeds := "Unit1.Em6.HmiInterface".cm.brakeTest.mendrelCathodeFrontAxisZ)
   END_RUNG
   // the same network as SCL:
   #instLER_BrakeTestMendrelCathodeFrontAxisZ(modeManual := "Unit1.EmNodes".unitStatus.mode.manual,   // "LER_BrakeTest"
                           modeMaintenance := "Unit1.EmNodes".unitStatus.mode.maintenance,
                           EnableManualCmds := #statEnableManualCmds,
                           mcRun := "Unit1.ControlNodes".motorPowerMC.run,
                           all_FdoorClose := "Unit1.EmNodes".AllFDoorClosed,
                           allDoorsOK := "Unit1.EmNodes".devicesSummary.allDoorsOK,
                           all_BrakeTest := #statAllBrakeTest.allStart,
                           hardwareId := "BA040AZSCU7~PROFINET_interface~BA040AZSDR28_SIEMENS_telegr,,,_2",
                           statUnitStatus := #statUnitStatus,
                           BrakeTestControlNoeds := "Unit1.Em6.ControlNodes".cm.brakeTest.mendrelCathodeFrontAxisZ,
                           axis_ControlNode := "Unit1.Em6.ControlNodes".cmMendrelCathodeFrontAxisZ,
                           axis_HmiInterface := "Unit1.Em6.HmiInterface".cmMendrelCathodeFrontAxisZ,
                           axis_Configuration := "Unit1.Em6.Config".cmMendrelCathodeFrontAxisZ,
                           HmiBrakeTestControlNoeds := "Unit1.Em6.HmiInterface".cm.brakeTest.mendrelCathodeFrontAxisZ);
END_REGION

REGION Network 303: Mendrel Cathode Rear Z-Axis Brake Test
   RUNG wire#powerrail
      #instLER_BrakeTestMendrelCathodeRearAxisZ(modeManual := "Unit1.EmNodes".unitStatus.mode.manual, modeMaintenance := "Unit1.EmNodes".unitStatus.mode.maintenance, EnableManualCmds := #statEnableManualCmds, mcRun := "Unit1.ControlNodes".motorPowerMC.run, all_FdoorClose := "Unit1.EmNodes".AllFDoorClosed, allDoorsOK := "Unit1.EmNodes".devicesSummary.allDoorsOK, all_BrakeTest := #statAllBrakeTest.allStart, hardwareId := "BA040AZSCU7~PROFINET_interface~BA040AZSDR30_SIEMENS_telegr,,,_2", statUnitStatus := #statUnitStatus, BrakeTestControlNoeds := "Unit1.Em6.ControlNodes".cm.brakeTest.mendrelCathodeRearAxisZ, axis_ControlNode := "Unit1.Em6.ControlNodes".cmMendrelCathodeRearAxisZ, axis_HmiInterface := "Unit1.Em6.HmiInterface".cmMendrelCathodeRearAxisZ, axis_Configuration := "Unit1.Em6.Config".cmMendrelCathodeRearAxisZ, HmiBrakeTestControlNoeds := "Unit1.Em6.HmiInterface".cm.brakeTest.mendrelCathodeRearAxisZ)
   END_RUNG
   // the same network as SCL:
   #instLER_BrakeTestMendrelCathodeRearAxisZ(modeManual := "Unit1.EmNodes".unitStatus.mode.manual,   // "LER_BrakeTest"
                           modeMaintenance := "Unit1.EmNodes".unitStatus.mode.maintenance,
                           EnableManualCmds := #statEnableManualCmds,
                           mcRun := "Unit1.ControlNodes".motorPowerMC.run,
                           all_FdoorClose := "Unit1.EmNodes".AllFDoorClosed,
                           allDoorsOK := "Unit1.EmNodes".devicesSummary.allDoorsOK,
                           all_BrakeTest := #statAllBrakeTest.allStart,
                           hardwareId := "BA040AZSCU7~PROFINET_interface~BA040AZSDR30_SIEMENS_telegr,,,_2",
                           statUnitStatus := #statUnitStatus,
                           BrakeTestControlNoeds := "Unit1.Em6.ControlNodes".cm.brakeTest.mendrelCathodeRearAxisZ,
                           axis_ControlNode := "Unit1.Em6.ControlNodes".cmMendrelCathodeRearAxisZ,
                           axis_HmiInterface := "Unit1.Em6.HmiInterface".cmMendrelCathodeRearAxisZ,
                           axis_Configuration := "Unit1.Em6.Config".cmMendrelCathodeRearAxisZ,
                           HmiBrakeTestControlNoeds := "Unit1.Em6.HmiInterface".cm.brakeTest.mendrelCathodeRearAxisZ);
END_REGION

REGION Network 304: Stack Table Z-Axis Brake Test
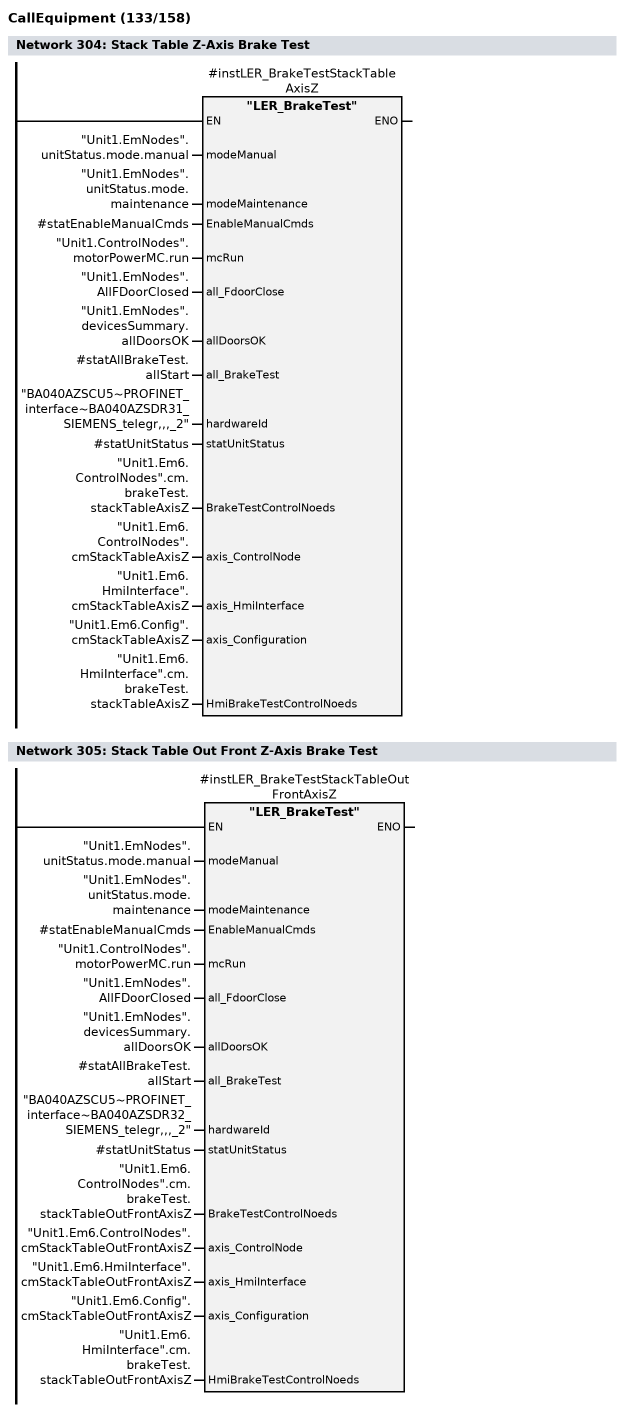
   RUNG wire#powerrail
      #instLER_BrakeTestStackTableAxisZ(modeManual := "Unit1.EmNodes".unitStatus.mode.manual, modeMaintenance := "Unit1.EmNodes".unitStatus.mode.maintenance, EnableManualCmds := #statEnableManualCmds, mcRun := "Unit1.ControlNodes".motorPowerMC.run, all_FdoorClose := "Unit1.EmNodes".AllFDoorClosed, allDoorsOK := "Unit1.EmNodes".devicesSummary.allDoorsOK, all_BrakeTest := #statAllBrakeTest.allStart, hardwareId := "BA040AZSCU5~PROFINET_interface~BA040AZSDR31_SIEMENS_telegr,,,_2", statUnitStatus := #statUnitStatus, BrakeTestControlNoeds := "Unit1.Em6.ControlNodes".cm.brakeTest.stackTableAxisZ, axis_ControlNode := "Unit1.Em6.ControlNodes".cmStackTableAxisZ, axis_HmiInterface := "Unit1.Em6.HmiInterface".cmStackTableAxisZ, axis_Configuration := "Unit1.Em6.Config".cmStackTableAxisZ, HmiBrakeTestControlNoeds := "Unit1.Em6.HmiInterface".cm.brakeTest.stackTableAxisZ)
   END_RUNG
   // the same network as SCL:
   #instLER_BrakeTestStackTableAxisZ(modeManual := "Unit1.EmNodes".unitStatus.mode.manual,   // "LER_BrakeTest"
                           modeMaintenance := "Unit1.EmNodes".unitStatus.mode.maintenance,
                           EnableManualCmds := #statEnableManualCmds,
                           mcRun := "Unit1.ControlNodes".motorPowerMC.run,
                           all_FdoorClose := "Unit1.EmNodes".AllFDoorClosed,
                           allDoorsOK := "Unit1.EmNodes".devicesSummary.allDoorsOK,
                           all_BrakeTest := #statAllBrakeTest.allStart,
                           hardwareId := "BA040AZSCU5~PROFINET_interface~BA040AZSDR31_SIEMENS_telegr,,,_2",
                           statUnitStatus := #statUnitStatus,
                           BrakeTestControlNoeds := "Unit1.Em6.ControlNodes".cm.brakeTest.stackTableAxisZ,
                           axis_ControlNode := "Unit1.Em6.ControlNodes".cmStackTableAxisZ,
                           axis_HmiInterface := "Unit1.Em6.HmiInterface".cmStackTableAxisZ,
                           axis_Configuration := "Unit1.Em6.Config".cmStackTableAxisZ,
                           HmiBrakeTestControlNoeds := "Unit1.Em6.HmiInterface".cm.brakeTest.stackTableAxisZ);
END_REGION

REGION Network 305: Stack Table Out Front Z-Axis Brake Test
   RUNG wire#powerrail
      #instLER_BrakeTestStackTableOutFrontAxisZ(modeManual := "Unit1.EmNodes".unitStatus.mode.manual, modeMaintenance := "Unit1.EmNodes".unitStatus.mode.maintenance, EnableManualCmds := #statEnableManualCmds, mcRun := "Unit1.ControlNodes".motorPowerMC.run, all_FdoorClose := "Unit1.EmNodes".AllFDoorClosed, allDoorsOK := "Unit1.EmNodes".devicesSummary.allDoorsOK, all_BrakeTest := #statAllBrakeTest.allStart, hardwareId := "BA040AZSCU5~PROFINET_interface~BA040AZSDR32_SIEMENS_telegr,,,_2", statUnitStatus := #statUnitStatus, BrakeTestControlNoeds := "Unit1.Em6.ControlNodes".cm.brakeTest.stackTableOutFrontAxisZ, axis_ControlNode := "Unit1.Em6.ControlNodes".cmStackTableOutFrontAxisZ, axis_HmiInterface := "Unit1.Em6.HmiInterface".cmStackTableOutFrontAxisZ, axis_Configuration := "Unit1.Em6.Config".cmStackTableOutFrontAxisZ, HmiBrakeTestControlNoeds := "Unit1.Em6.HmiInterface".cm.brakeTest.stackTableOutFrontAxisZ)
   END_RUNG
   // the same network as SCL:
   #instLER_BrakeTestStackTableOutFrontAxisZ(modeManual := "Unit1.EmNodes".unitStatus.mode.manual,   // "LER_BrakeTest"
                           modeMaintenance := "Unit1.EmNodes".unitStatus.mode.maintenance,
                           EnableManualCmds := #statEnableManualCmds,
                           mcRun := "Unit1.ControlNodes".motorPowerMC.run,
                           all_FdoorClose := "Unit1.EmNodes".AllFDoorClosed,
                           allDoorsOK := "Unit1.EmNodes".devicesSummary.allDoorsOK,
                           all_BrakeTest := #statAllBrakeTest.allStart,
                           hardwareId := "BA040AZSCU5~PROFINET_interface~BA040AZSDR32_SIEMENS_telegr,,,_2",
                           statUnitStatus := #statUnitStatus,
                           BrakeTestControlNoeds := "Unit1.Em6.ControlNodes".cm.brakeTest.stackTableOutFrontAxisZ,
                           axis_ControlNode := "Unit1.Em6.ControlNodes".cmStackTableOutFrontAxisZ,
                           axis_HmiInterface := "Unit1.Em6.HmiInterface".cmStackTableOutFrontAxisZ,
                           axis_Configuration := "Unit1.Em6.Config".cmStackTableOutFrontAxisZ,
                           HmiBrakeTestControlNoeds := "Unit1.Em6.HmiInterface".cm.brakeTest.stackTableOutFrontAxisZ);
END_REGION

REGION Network 306: Stack Table Out Rear Z-Axis Brake Test
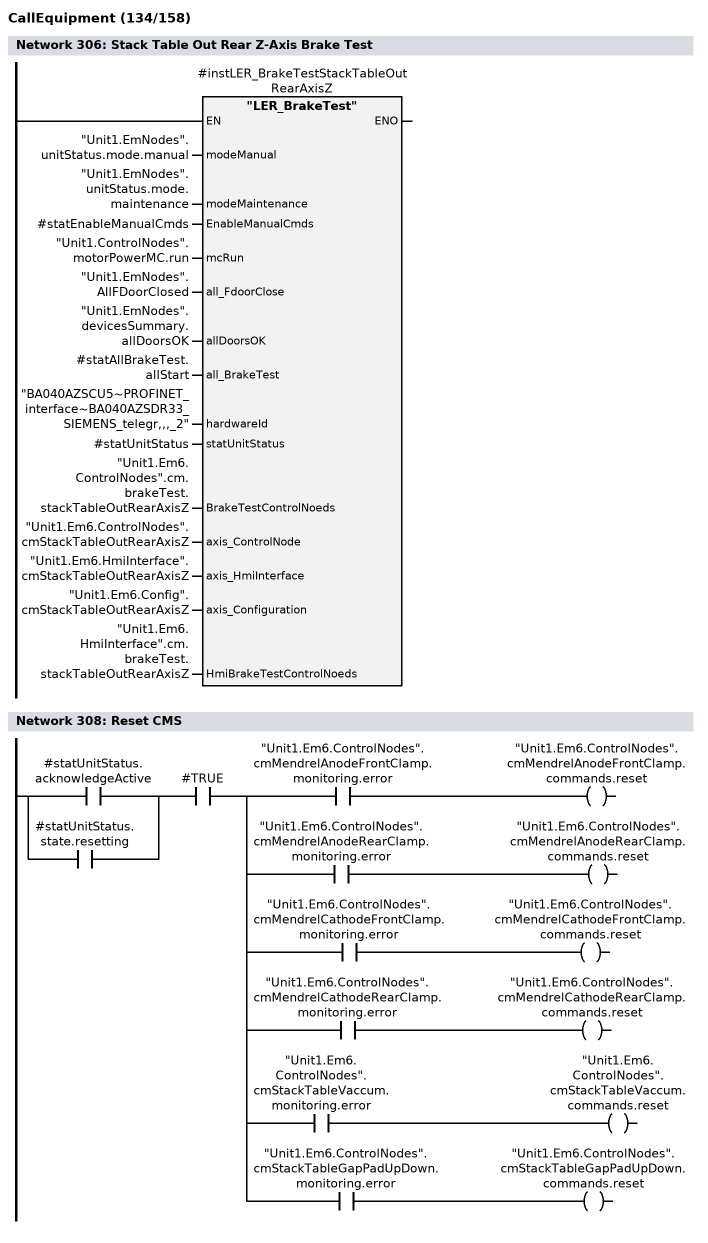
   RUNG wire#powerrail
      #instLER_BrakeTestStackTableOutRearAxisZ(modeManual := "Unit1.EmNodes".unitStatus.mode.manual, modeMaintenance := "Unit1.EmNodes".unitStatus.mode.maintenance, EnableManualCmds := #statEnableManualCmds, mcRun := "Unit1.ControlNodes".motorPowerMC.run, all_FdoorClose := "Unit1.EmNodes".AllFDoorClosed, allDoorsOK := "Unit1.EmNodes".devicesSummary.allDoorsOK, all_BrakeTest := #statAllBrakeTest.allStart, hardwareId := "BA040AZSCU5~PROFINET_interface~BA040AZSDR33_SIEMENS_telegr,,,_2", statUnitStatus := #statUnitStatus, BrakeTestControlNoeds := "Unit1.Em6.ControlNodes".cm.brakeTest.stackTableOutRearAxisZ, axis_ControlNode := "Unit1.Em6.ControlNodes".cmStackTableOutRearAxisZ, axis_HmiInterface := "Unit1.Em6.HmiInterface".cmStackTableOutRearAxisZ, axis_Configuration := "Unit1.Em6.Config".cmStackTableOutRearAxisZ, HmiBrakeTestControlNoeds := "Unit1.Em6.HmiInterface".cm.brakeTest.stackTableOutRearAxisZ)
   END_RUNG
   // the same network as SCL:
   #instLER_BrakeTestStackTableOutRearAxisZ(modeManual := "Unit1.EmNodes".unitStatus.mode.manual,   // "LER_BrakeTest"
                           modeMaintenance := "Unit1.EmNodes".unitStatus.mode.maintenance,
                           EnableManualCmds := #statEnableManualCmds,
                           mcRun := "Unit1.ControlNodes".motorPowerMC.run,
                           all_FdoorClose := "Unit1.EmNodes".AllFDoorClosed,
                           allDoorsOK := "Unit1.EmNodes".devicesSummary.allDoorsOK,
                           all_BrakeTest := #statAllBrakeTest.allStart,
                           hardwareId := "BA040AZSCU5~PROFINET_interface~BA040AZSDR33_SIEMENS_telegr,,,_2",
                           statUnitStatus := #statUnitStatus,
                           BrakeTestControlNoeds := "Unit1.Em6.ControlNodes".cm.brakeTest.stackTableOutRearAxisZ,
                           axis_ControlNode := "Unit1.Em6.ControlNodes".cmStackTableOutRearAxisZ,
                           axis_HmiInterface := "Unit1.Em6.HmiInterface".cmStackTableOutRearAxisZ,
                           axis_Configuration := "Unit1.Em6.Config".cmStackTableOutRearAxisZ,
                           HmiBrakeTestControlNoeds := "Unit1.Em6.HmiInterface".cm.brakeTest.stackTableOutRearAxisZ);
END_REGION

REGION Network 307: ********** Control Modules (TwoWayActuator) **********
END_REGION

REGION Network 308: Reset CMS
   RUNG wire#powerrail
      Contact( #statUnitStatus.acknowledgeActive )
      wire#w1
      Contact( #TRUE )
      wire#w2
      Contact( "Unit1.Em6.ControlNodes".cmMendrelAnodeFrontClamp.monitoring.error )
      Coil( "Unit1.Em6.ControlNodes".cmMendrelAnodeFrontClamp.commands.reset )
   END_RUNG
   RUNG wire#powerrail
      Contact( #statUnitStatus.state.resetting )
   END_RUNG wire#w1
   RUNG wire#w2
      Contact( "Unit1.Em6.ControlNodes".cmMendrelAnodeRearClamp.monitoring.error )
      Coil( "Unit1.Em6.ControlNodes".cmMendrelAnodeRearClamp.commands.reset )
   END_RUNG
   RUNG wire#w2
      Contact( "Unit1.Em6.ControlNodes".cmMendrelCathodeFrontClamp.monitoring.error )
      Coil( "Unit1.Em6.ControlNodes".cmMendrelCathodeFrontClamp.commands.reset )
   END_RUNG
   RUNG wire#w2
      Contact( "Unit1.Em6.ControlNodes".cmMendrelCathodeRearClamp.monitoring.error )
      Coil( "Unit1.Em6.ControlNodes".cmMendrelCathodeRearClamp.commands.reset )
   END_RUNG
   RUNG wire#w2
      Contact( "Unit1.Em6.ControlNodes".cmStackTableVaccum.monitoring.error )
      Coil( "Unit1.Em6.ControlNodes".cmStackTableVaccum.commands.reset )
   END_RUNG
   RUNG wire#w2
      Contact( "Unit1.Em6.ControlNodes".cmStackTableGapPadUpDown.monitoring.error )
      Coil( "Unit1.Em6.ControlNodes".cmStackTableGapPadUpDown.commands.reset )
   END_RUNG
   // the same network as SCL:
   #_w1 := (#statUnitStatus.acknowledgeActive OR #statUnitStatus.state.resetting) AND #TRUE;
   "Unit1.Em6.ControlNodes".cmMendrelAnodeFrontClamp.commands.reset := #_w1 AND "Unit1.Em6.ControlNodes".cmMendrelAnodeFrontClamp.monitoring.error;
   "Unit1.Em6.ControlNodes".cmMendrelAnodeRearClamp.commands.reset := #_w1 AND "Unit1.Em6.ControlNodes".cmMendrelAnodeRearClamp.monitoring.error;
   "Unit1.Em6.ControlNodes".cmMendrelCathodeFrontClamp.commands.reset := #_w1 AND "Unit1.Em6.ControlNodes".cmMendrelCathodeFrontClamp.monitoring.error;
   "Unit1.Em6.ControlNodes".cmMendrelCathodeRearClamp.commands.reset := #_w1 AND "Unit1.Em6.ControlNodes".cmMendrelCathodeRearClamp.monitoring.error;
   "Unit1.Em6.ControlNodes".cmStackTableVaccum.commands.reset := #_w1 AND "Unit1.Em6.ControlNodes".cmStackTableVaccum.monitoring.error;
   "Unit1.Em6.ControlNodes".cmStackTableGapPadUpDown.commands.reset := #_w1 AND "Unit1.Em6.ControlNodes".cmStackTableGapPadUpDown.monitoring.error;
END_REGION

REGION Network 310: CmMendrelAnodeFrontClamp Interlock
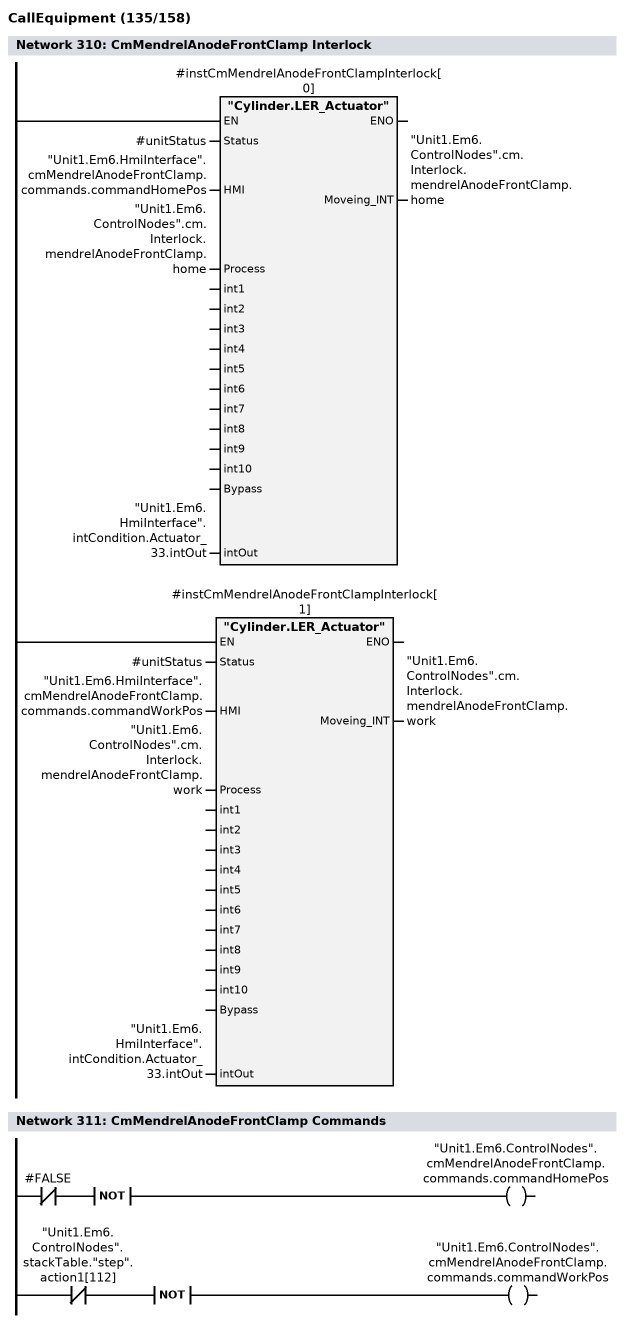
   RUNG wire#powerrail
      #instCmMendrelAnodeFrontClampInterlock[0](Status := #unitStatus, HMI := "Unit1.Em6.HmiInterface".cmMendrelAnodeFrontClamp.commands.commandHomePos, Process := "Unit1.Em6.ControlNodes".cm.Interlock.mendrelAnodeFrontClamp.home, int1 :=, int2 :=, int3 :=, int4 :=, int5 :=, int6 :=, int7 :=, int8 :=, int9 :=, int10 :=, Bypass :=, intOut := "Unit1.Em6.HmiInterface".intCondition.Actuator_33.intOut, Moveing_INT => "Unit1.Em6.ControlNodes".cm.Interlock.mendrelAnodeFrontClamp.home)
   END_RUNG
   RUNG wire#powerrail
      #instCmMendrelAnodeFrontClampInterlock[1](Status := #unitStatus, HMI := "Unit1.Em6.HmiInterface".cmMendrelAnodeFrontClamp.commands.commandWorkPos, Process := "Unit1.Em6.ControlNodes".cm.Interlock.mendrelAnodeFrontClamp.work, int1 :=, int2 :=, int3 :=, int4 :=, int5 :=, int6 :=, int7 :=, int8 :=, int9 :=, int10 :=, Bypass :=, intOut := "Unit1.Em6.HmiInterface".intCondition.Actuator_33.intOut, Moveing_INT => "Unit1.Em6.ControlNodes".cm.Interlock.mendrelAnodeFrontClamp.work)
   END_RUNG
   // the same network as SCL:
   #instCmMendrelAnodeFrontClampInterlock[0](Status := #unitStatus,   // "Cylinder.LER_Actuator"
                           HMI := "Unit1.Em6.HmiInterface".cmMendrelAnodeFrontClamp.commands.commandHomePos,
                           Process := "Unit1.Em6.ControlNodes".cm.Interlock.mendrelAnodeFrontClamp.home,
                           intOut := "Unit1.Em6.HmiInterface".intCondition.Actuator_33.intOut,
                           Moveing_INT => "Unit1.Em6.ControlNodes".cm.Interlock.mendrelAnodeFrontClamp.home);
   #instCmMendrelAnodeFrontClampInterlock[1](Status := #unitStatus,   // "Cylinder.LER_Actuator"
                           HMI := "Unit1.Em6.HmiInterface".cmMendrelAnodeFrontClamp.commands.commandWorkPos,
                           Process := "Unit1.Em6.ControlNodes".cm.Interlock.mendrelAnodeFrontClamp.work,
                           intOut := "Unit1.Em6.HmiInterface".intCondition.Actuator_33.intOut,
                           Moveing_INT => "Unit1.Em6.ControlNodes".cm.Interlock.mendrelAnodeFrontClamp.work);
END_REGION

REGION Network 311: CmMendrelAnodeFrontClamp Commands
   RUNG wire#powerrail
      I_Contact( #FALSE )
      Not()
      Coil( "Unit1.Em6.ControlNodes".cmMendrelAnodeFrontClamp.commands.commandHomePos )
   END_RUNG
   RUNG wire#powerrail
      I_Contact( "Unit1.Em6.ControlNodes".stackTable."step".action1[112] )
      Not()
      Coil( "Unit1.Em6.ControlNodes".cmMendrelAnodeFrontClamp.commands.commandWorkPos )
   END_RUNG
   // the same network as SCL:
   "Unit1.Em6.ControlNodes".cmMendrelAnodeFrontClamp.commands.commandHomePos := NOT (NOT #FALSE);
   "Unit1.Em6.ControlNodes".cmMendrelAnodeFrontClamp.commands.commandWorkPos := NOT (NOT "Unit1.Em6.ControlNodes".stackTable."step".action1[112]);
END_REGION

REGION Network 312: Call instCmMendrelAnodeFrontClamp
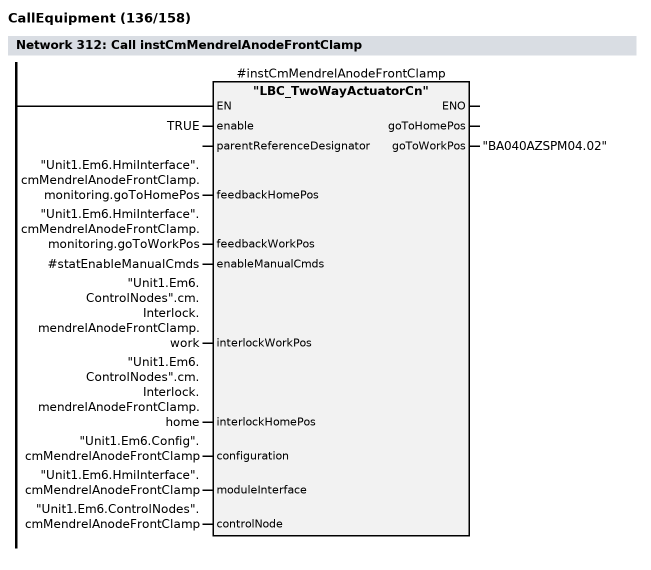
   RUNG wire#powerrail
      #instCmMendrelAnodeFrontClamp(enable := TRUE, parentReferenceDesignator :=, feedbackHomePos := "Unit1.Em6.HmiInterface".cmMendrelAnodeFrontClamp.monitoring.goToHomePos, feedbackWorkPos := "Unit1.Em6.HmiInterface".cmMendrelAnodeFrontClamp.monitoring.goToWorkPos, enableManualCmds := #statEnableManualCmds, interlockWorkPos := "Unit1.Em6.ControlNodes".cm.Interlock.mendrelAnodeFrontClamp.work, interlockHomePos := "Unit1.Em6.ControlNodes".cm.Interlock.mendrelAnodeFrontClamp.home, configuration := "Unit1.Em6.Config".cmMendrelAnodeFrontClamp, moduleInterface := "Unit1.Em6.HmiInterface".cmMendrelAnodeFrontClamp, controlNode := "Unit1.Em6.ControlNodes".cmMendrelAnodeFrontClamp, goToHomePos =>, goToWorkPos => "BA040AZSPM04.02")
   END_RUNG
   // the same network as SCL:
   #instCmMendrelAnodeFrontClamp(enable := TRUE,   // "LBC_TwoWayActuatorCn"
                           feedbackHomePos := "Unit1.Em6.HmiInterface".cmMendrelAnodeFrontClamp.monitoring.goToHomePos,
                           feedbackWorkPos := "Unit1.Em6.HmiInterface".cmMendrelAnodeFrontClamp.monitoring.goToWorkPos,
                           enableManualCmds := #statEnableManualCmds,
                           interlockWorkPos := "Unit1.Em6.ControlNodes".cm.Interlock.mendrelAnodeFrontClamp.work,
                           interlockHomePos := "Unit1.Em6.ControlNodes".cm.Interlock.mendrelAnodeFrontClamp.home,
                           configuration := "Unit1.Em6.Config".cmMendrelAnodeFrontClamp,
                           moduleInterface := "Unit1.Em6.HmiInterface".cmMendrelAnodeFrontClamp,
                           controlNode := "Unit1.Em6.ControlNodes".cmMendrelAnodeFrontClamp,
                           goToWorkPos => "BA040AZSPM04.02");
END_REGION

REGION Network 314: CmMendrelAnodeRearClamp Interlock
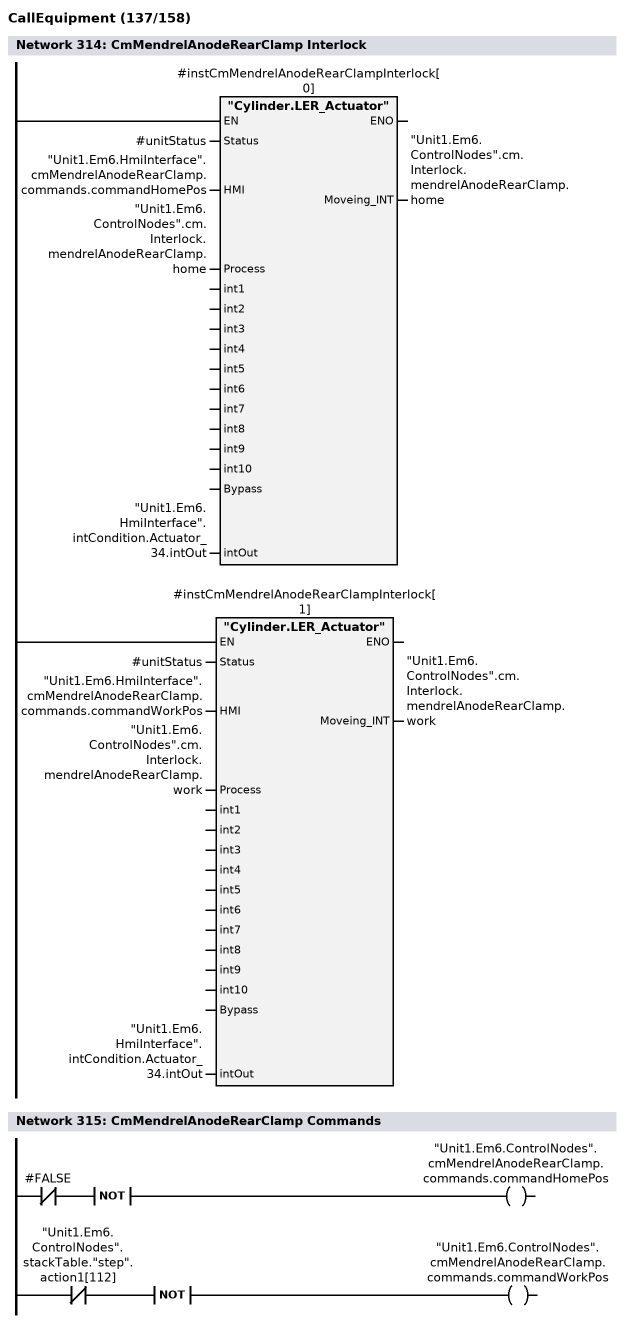
   RUNG wire#powerrail
      #instCmMendrelAnodeRearClampInterlock[0](Status := #unitStatus, HMI := "Unit1.Em6.HmiInterface".cmMendrelAnodeRearClamp.commands.commandHomePos, Process := "Unit1.Em6.ControlNodes".cm.Interlock.mendrelAnodeRearClamp.home, int1 :=, int2 :=, int3 :=, int4 :=, int5 :=, int6 :=, int7 :=, int8 :=, int9 :=, int10 :=, Bypass :=, intOut := "Unit1.Em6.HmiInterface".intCondition.Actuator_34.intOut, Moveing_INT => "Unit1.Em6.ControlNodes".cm.Interlock.mendrelAnodeRearClamp.home)
   END_RUNG
   RUNG wire#powerrail
      #instCmMendrelAnodeRearClampInterlock[1](Status := #unitStatus, HMI := "Unit1.Em6.HmiInterface".cmMendrelAnodeRearClamp.commands.commandWorkPos, Process := "Unit1.Em6.ControlNodes".cm.Interlock.mendrelAnodeRearClamp.work, int1 :=, int2 :=, int3 :=, int4 :=, int5 :=, int6 :=, int7 :=, int8 :=, int9 :=, int10 :=, Bypass :=, intOut := "Unit1.Em6.HmiInterface".intCondition.Actuator_34.intOut, Moveing_INT => "Unit1.Em6.ControlNodes".cm.Interlock.mendrelAnodeRearClamp.work)
   END_RUNG
   // the same network as SCL:
   #instCmMendrelAnodeRearClampInterlock[0](Status := #unitStatus,   // "Cylinder.LER_Actuator"
                           HMI := "Unit1.Em6.HmiInterface".cmMendrelAnodeRearClamp.commands.commandHomePos,
                           Process := "Unit1.Em6.ControlNodes".cm.Interlock.mendrelAnodeRearClamp.home,
                           intOut := "Unit1.Em6.HmiInterface".intCondition.Actuator_34.intOut,
                           Moveing_INT => "Unit1.Em6.ControlNodes".cm.Interlock.mendrelAnodeRearClamp.home);
   #instCmMendrelAnodeRearClampInterlock[1](Status := #unitStatus,   // "Cylinder.LER_Actuator"
                           HMI := "Unit1.Em6.HmiInterface".cmMendrelAnodeRearClamp.commands.commandWorkPos,
                           Process := "Unit1.Em6.ControlNodes".cm.Interlock.mendrelAnodeRearClamp.work,
                           intOut := "Unit1.Em6.HmiInterface".intCondition.Actuator_34.intOut,
                           Moveing_INT => "Unit1.Em6.ControlNodes".cm.Interlock.mendrelAnodeRearClamp.work);
END_REGION

REGION Network 315: CmMendrelAnodeRearClamp Commands
   RUNG wire#powerrail
      I_Contact( #FALSE )
      Not()
      Coil( "Unit1.Em6.ControlNodes".cmMendrelAnodeRearClamp.commands.commandHomePos )
   END_RUNG
   RUNG wire#powerrail
      I_Contact( "Unit1.Em6.ControlNodes".stackTable."step".action1[112] )
      Not()
      Coil( "Unit1.Em6.ControlNodes".cmMendrelAnodeRearClamp.commands.commandWorkPos )
   END_RUNG
   // the same network as SCL:
   "Unit1.Em6.ControlNodes".cmMendrelAnodeRearClamp.commands.commandHomePos := NOT (NOT #FALSE);
   "Unit1.Em6.ControlNodes".cmMendrelAnodeRearClamp.commands.commandWorkPos := NOT (NOT "Unit1.Em6.ControlNodes".stackTable."step".action1[112]);
END_REGION

REGION Network 316: Call instCmMendrelAnodeRearClamp
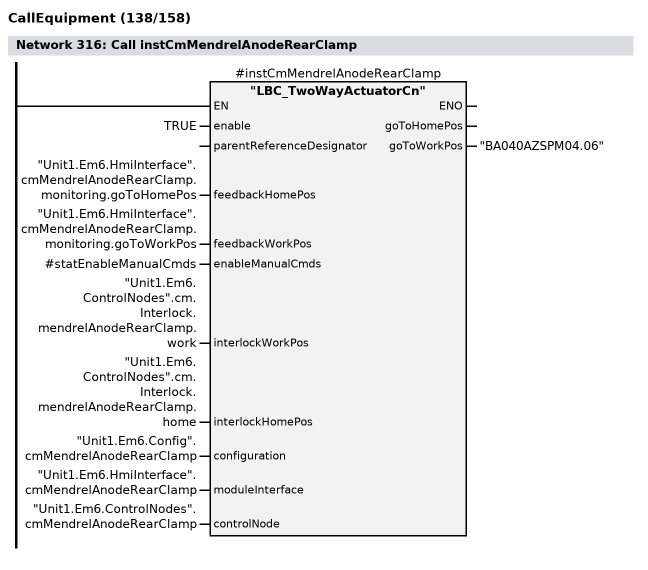
   RUNG wire#powerrail
      #instCmMendrelAnodeRearClamp(enable := TRUE, parentReferenceDesignator :=, feedbackHomePos := "Unit1.Em6.HmiInterface".cmMendrelAnodeRearClamp.monitoring.goToHomePos, feedbackWorkPos := "Unit1.Em6.HmiInterface".cmMendrelAnodeRearClamp.monitoring.goToWorkPos, enableManualCmds := #statEnableManualCmds, interlockWorkPos := "Unit1.Em6.ControlNodes".cm.Interlock.mendrelAnodeRearClamp.work, interlockHomePos := "Unit1.Em6.ControlNodes".cm.Interlock.mendrelAnodeRearClamp.home, configuration := "Unit1.Em6.Config".cmMendrelAnodeRearClamp, moduleInterface := "Unit1.Em6.HmiInterface".cmMendrelAnodeRearClamp, controlNode := "Unit1.Em6.ControlNodes".cmMendrelAnodeRearClamp, goToHomePos =>, goToWorkPos => "BA040AZSPM04.06")
   END_RUNG
   // the same network as SCL:
   #instCmMendrelAnodeRearClamp(enable := TRUE,   // "LBC_TwoWayActuatorCn"
                           feedbackHomePos := "Unit1.Em6.HmiInterface".cmMendrelAnodeRearClamp.monitoring.goToHomePos,
                           feedbackWorkPos := "Unit1.Em6.HmiInterface".cmMendrelAnodeRearClamp.monitoring.goToWorkPos,
                           enableManualCmds := #statEnableManualCmds,
                           interlockWorkPos := "Unit1.Em6.ControlNodes".cm.Interlock.mendrelAnodeRearClamp.work,
                           interlockHomePos := "Unit1.Em6.ControlNodes".cm.Interlock.mendrelAnodeRearClamp.home,
                           configuration := "Unit1.Em6.Config".cmMendrelAnodeRearClamp,
                           moduleInterface := "Unit1.Em6.HmiInterface".cmMendrelAnodeRearClamp,
                           controlNode := "Unit1.Em6.ControlNodes".cmMendrelAnodeRearClamp,
                           goToWorkPos => "BA040AZSPM04.06");
END_REGION

REGION Network 318: CmMendrelCathodeFrontClamp Interlock
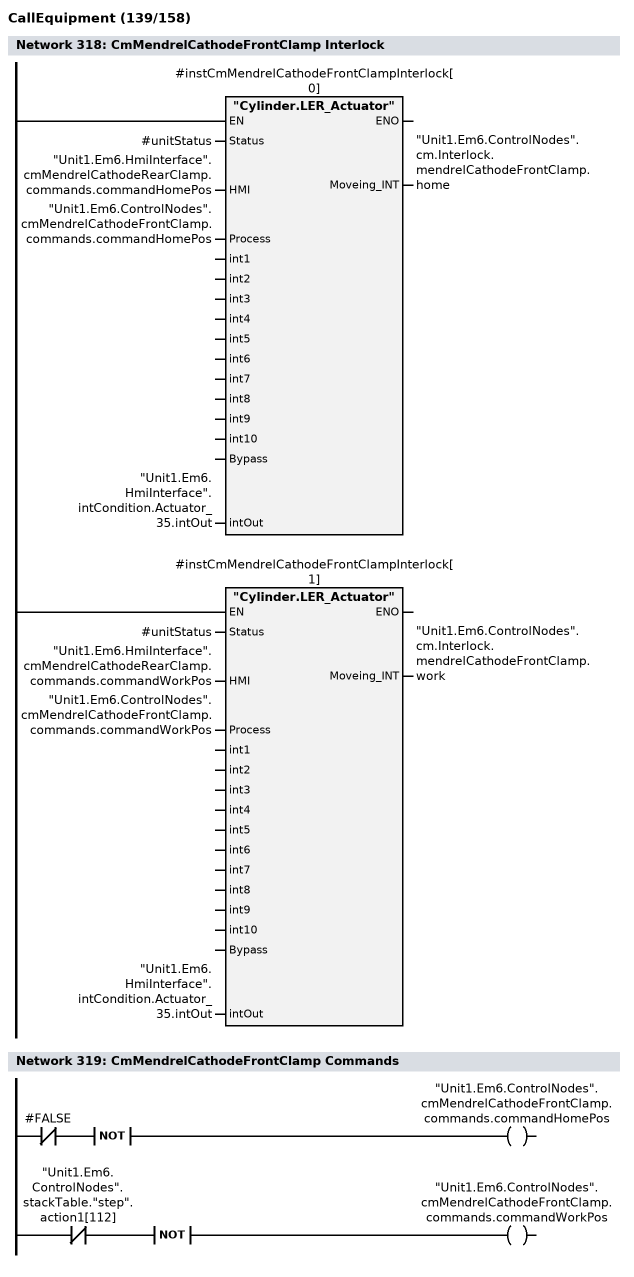
   RUNG wire#powerrail
      #instCmMendrelCathodeFrontClampInterlock[0](Status := #unitStatus, HMI := "Unit1.Em6.HmiInterface".cmMendrelCathodeRearClamp.commands.commandHomePos, Process := "Unit1.Em6.ControlNodes".cmMendrelCathodeFrontClamp.commands.commandHomePos, int1 :=, int2 :=, int3 :=, int4 :=, int5 :=, int6 :=, int7 :=, int8 :=, int9 :=, int10 :=, Bypass :=, intOut := "Unit1.Em6.HmiInterface".intCondition.Actuator_35.intOut, Moveing_INT => "Unit1.Em6.ControlNodes".cm.Interlock.mendrelCathodeFrontClamp.home)
   END_RUNG
   RUNG wire#powerrail
      #instCmMendrelCathodeFrontClampInterlock[1](Status := #unitStatus, HMI := "Unit1.Em6.HmiInterface".cmMendrelCathodeRearClamp.commands.commandWorkPos, Process := "Unit1.Em6.ControlNodes".cmMendrelCathodeFrontClamp.commands.commandWorkPos, int1 :=, int2 :=, int3 :=, int4 :=, int5 :=, int6 :=, int7 :=, int8 :=, int9 :=, int10 :=, Bypass :=, intOut := "Unit1.Em6.HmiInterface".intCondition.Actuator_35.intOut, Moveing_INT => "Unit1.Em6.ControlNodes".cm.Interlock.mendrelCathodeFrontClamp.work)
   END_RUNG
   // the same network as SCL:
   #instCmMendrelCathodeFrontClampInterlock[0](Status := #unitStatus,   // "Cylinder.LER_Actuator"
                           HMI := "Unit1.Em6.HmiInterface".cmMendrelCathodeRearClamp.commands.commandHomePos,
                           Process := "Unit1.Em6.ControlNodes".cmMendrelCathodeFrontClamp.commands.commandHomePos,
                           intOut := "Unit1.Em6.HmiInterface".intCondition.Actuator_35.intOut,
                           Moveing_INT => "Unit1.Em6.ControlNodes".cm.Interlock.mendrelCathodeFrontClamp.home);
   #instCmMendrelCathodeFrontClampInterlock[1](Status := #unitStatus,   // "Cylinder.LER_Actuator"
                           HMI := "Unit1.Em6.HmiInterface".cmMendrelCathodeRearClamp.commands.commandWorkPos,
                           Process := "Unit1.Em6.ControlNodes".cmMendrelCathodeFrontClamp.commands.commandWorkPos,
                           intOut := "Unit1.Em6.HmiInterface".intCondition.Actuator_35.intOut,
                           Moveing_INT => "Unit1.Em6.ControlNodes".cm.Interlock.mendrelCathodeFrontClamp.work);
END_REGION

REGION Network 319: CmMendrelCathodeFrontClamp Commands
   RUNG wire#powerrail
      I_Contact( #FALSE )
      Not()
      Coil( "Unit1.Em6.ControlNodes".cmMendrelCathodeFrontClamp.commands.commandHomePos )
   END_RUNG
   RUNG wire#powerrail
      I_Contact( "Unit1.Em6.ControlNodes".stackTable."step".action1[112] )
      Not()
      Coil( "Unit1.Em6.ControlNodes".cmMendrelCathodeFrontClamp.commands.commandWorkPos )
   END_RUNG
   // the same network as SCL:
   "Unit1.Em6.ControlNodes".cmMendrelCathodeFrontClamp.commands.commandHomePos := NOT (NOT #FALSE);
   "Unit1.Em6.ControlNodes".cmMendrelCathodeFrontClamp.commands.commandWorkPos := NOT (NOT "Unit1.Em6.ControlNodes".stackTable."step".action1[112]);
END_REGION

REGION Network 320: Call instCmMendrelCathodeFrontClamp
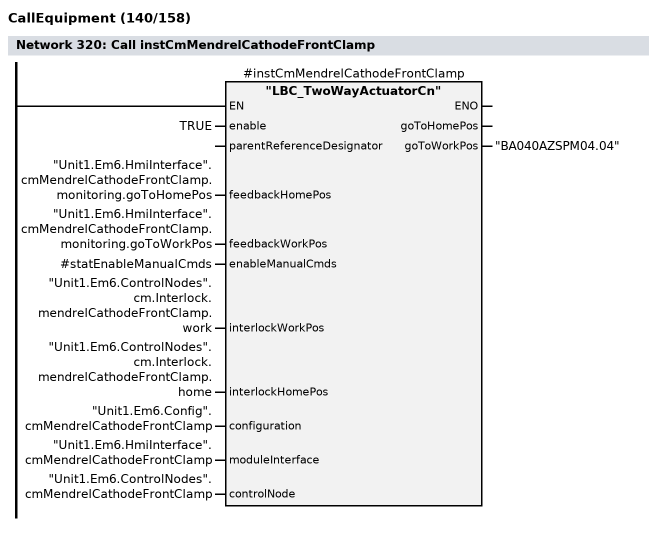
   RUNG wire#powerrail
      #instCmMendrelCathodeFrontClamp(enable := TRUE, parentReferenceDesignator :=, feedbackHomePos := "Unit1.Em6.HmiInterface".cmMendrelCathodeFrontClamp.monitoring.goToHomePos, feedbackWorkPos := "Unit1.Em6.HmiInterface".cmMendrelCathodeFrontClamp.monitoring.goToWorkPos, enableManualCmds := #statEnableManualCmds, interlockWorkPos := "Unit1.Em6.ControlNodes".cm.Interlock.mendrelCathodeFrontClamp.work, interlockHomePos := "Unit1.Em6.ControlNodes".cm.Interlock.mendrelCathodeFrontClamp.home, configuration := "Unit1.Em6.Config".cmMendrelCathodeFrontClamp, moduleInterface := "Unit1.Em6.HmiInterface".cmMendrelCathodeFrontClamp, controlNode := "Unit1.Em6.ControlNodes".cmMendrelCathodeFrontClamp, goToHomePos =>, goToWorkPos => "BA040AZSPM04.04")
   END_RUNG
   // the same network as SCL:
   #instCmMendrelCathodeFrontClamp(enable := TRUE,   // "LBC_TwoWayActuatorCn"
                           feedbackHomePos := "Unit1.Em6.HmiInterface".cmMendrelCathodeFrontClamp.monitoring.goToHomePos,
                           feedbackWorkPos := "Unit1.Em6.HmiInterface".cmMendrelCathodeFrontClamp.monitoring.goToWorkPos,
                           enableManualCmds := #statEnableManualCmds,
                           interlockWorkPos := "Unit1.Em6.ControlNodes".cm.Interlock.mendrelCathodeFrontClamp.work,
                           interlockHomePos := "Unit1.Em6.ControlNodes".cm.Interlock.mendrelCathodeFrontClamp.home,
                           configuration := "Unit1.Em6.Config".cmMendrelCathodeFrontClamp,
                           moduleInterface := "Unit1.Em6.HmiInterface".cmMendrelCathodeFrontClamp,
                           controlNode := "Unit1.Em6.ControlNodes".cmMendrelCathodeFrontClamp,
                           goToWorkPos => "BA040AZSPM04.04");
END_REGION

REGION Network 322: CmMendrelCathodeRearClamp Interlock
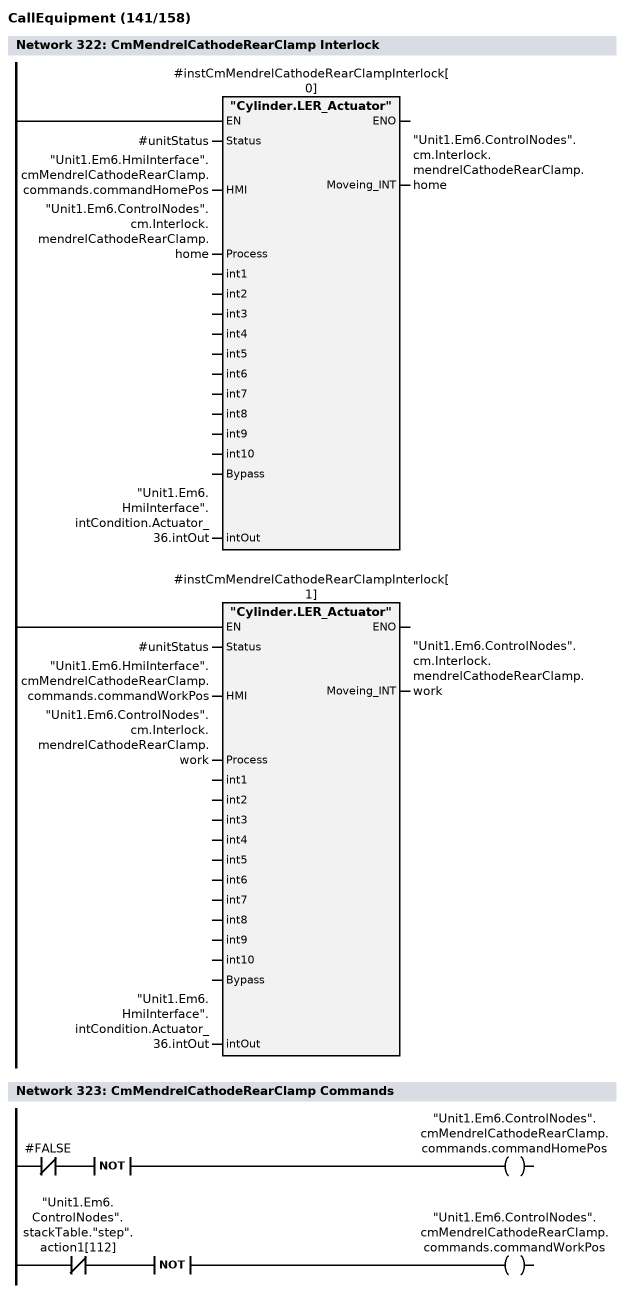
   RUNG wire#powerrail
      #instCmMendrelCathodeRearClampInterlock[0](Status := #unitStatus, HMI := "Unit1.Em6.HmiInterface".cmMendrelCathodeRearClamp.commands.commandHomePos, Process := "Unit1.Em6.ControlNodes".cm.Interlock.mendrelCathodeRearClamp.home, int1 :=, int2 :=, int3 :=, int4 :=, int5 :=, int6 :=, int7 :=, int8 :=, int9 :=, int10 :=, Bypass :=, intOut := "Unit1.Em6.HmiInterface".intCondition.Actuator_36.intOut, Moveing_INT => "Unit1.Em6.ControlNodes".cm.Interlock.mendrelCathodeRearClamp.home)
   END_RUNG
   RUNG wire#powerrail
      #instCmMendrelCathodeRearClampInterlock[1](Status := #unitStatus, HMI := "Unit1.Em6.HmiInterface".cmMendrelCathodeRearClamp.commands.commandWorkPos, Process := "Unit1.Em6.ControlNodes".cm.Interlock.mendrelCathodeRearClamp.work, int1 :=, int2 :=, int3 :=, int4 :=, int5 :=, int6 :=, int7 :=, int8 :=, int9 :=, int10 :=, Bypass :=, intOut := "Unit1.Em6.HmiInterface".intCondition.Actuator_36.intOut, Moveing_INT => "Unit1.Em6.ControlNodes".cm.Interlock.mendrelCathodeRearClamp.work)
   END_RUNG
   // the same network as SCL:
   #instCmMendrelCathodeRearClampInterlock[0](Status := #unitStatus,   // "Cylinder.LER_Actuator"
                           HMI := "Unit1.Em6.HmiInterface".cmMendrelCathodeRearClamp.commands.commandHomePos,
                           Process := "Unit1.Em6.ControlNodes".cm.Interlock.mendrelCathodeRearClamp.home,
                           intOut := "Unit1.Em6.HmiInterface".intCondition.Actuator_36.intOut,
                           Moveing_INT => "Unit1.Em6.ControlNodes".cm.Interlock.mendrelCathodeRearClamp.home);
   #instCmMendrelCathodeRearClampInterlock[1](Status := #unitStatus,   // "Cylinder.LER_Actuator"
                           HMI := "Unit1.Em6.HmiInterface".cmMendrelCathodeRearClamp.commands.commandWorkPos,
                           Process := "Unit1.Em6.ControlNodes".cm.Interlock.mendrelCathodeRearClamp.work,
                           intOut := "Unit1.Em6.HmiInterface".intCondition.Actuator_36.intOut,
                           Moveing_INT => "Unit1.Em6.ControlNodes".cm.Interlock.mendrelCathodeRearClamp.work);
END_REGION

REGION Network 323: CmMendrelCathodeRearClamp Commands
   RUNG wire#powerrail
      I_Contact( #FALSE )
      Not()
      Coil( "Unit1.Em6.ControlNodes".cmMendrelCathodeRearClamp.commands.commandHomePos )
   END_RUNG
   RUNG wire#powerrail
      I_Contact( "Unit1.Em6.ControlNodes".stackTable."step".action1[112] )
      Not()
      Coil( "Unit1.Em6.ControlNodes".cmMendrelCathodeRearClamp.commands.commandWorkPos )
   END_RUNG
   // the same network as SCL:
   "Unit1.Em6.ControlNodes".cmMendrelCathodeRearClamp.commands.commandHomePos := NOT (NOT #FALSE);
   "Unit1.Em6.ControlNodes".cmMendrelCathodeRearClamp.commands.commandWorkPos := NOT (NOT "Unit1.Em6.ControlNodes".stackTable."step".action1[112]);
END_REGION

REGION Network 324: Call instCmMendrelCathodeRearClamp
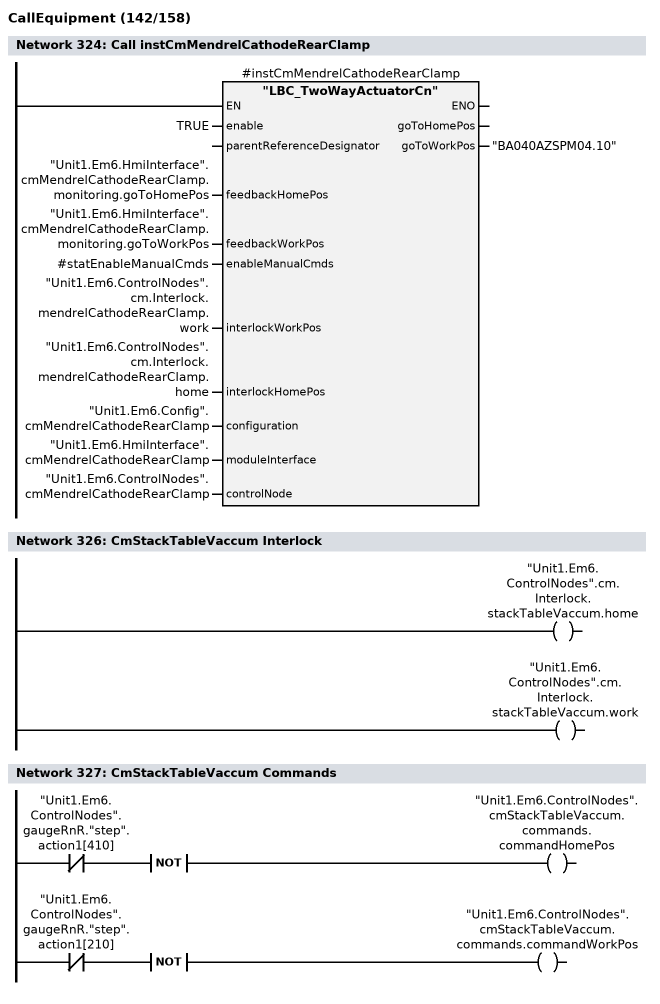
   RUNG wire#powerrail
      #instCmMendrelCathodeRearClamp(enable := TRUE, parentReferenceDesignator :=, feedbackHomePos := "Unit1.Em6.HmiInterface".cmMendrelCathodeRearClamp.monitoring.goToHomePos, feedbackWorkPos := "Unit1.Em6.HmiInterface".cmMendrelCathodeRearClamp.monitoring.goToWorkPos, enableManualCmds := #statEnableManualCmds, interlockWorkPos := "Unit1.Em6.ControlNodes".cm.Interlock.mendrelCathodeRearClamp.work, interlockHomePos := "Unit1.Em6.ControlNodes".cm.Interlock.mendrelCathodeRearClamp.home, configuration := "Unit1.Em6.Config".cmMendrelCathodeRearClamp, moduleInterface := "Unit1.Em6.HmiInterface".cmMendrelCathodeRearClamp, controlNode := "Unit1.Em6.ControlNodes".cmMendrelCathodeRearClamp, goToHomePos =>, goToWorkPos => "BA040AZSPM04.10")
   END_RUNG
   // the same network as SCL:
   #instCmMendrelCathodeRearClamp(enable := TRUE,   // "LBC_TwoWayActuatorCn"
                           feedbackHomePos := "Unit1.Em6.HmiInterface".cmMendrelCathodeRearClamp.monitoring.goToHomePos,
                           feedbackWorkPos := "Unit1.Em6.HmiInterface".cmMendrelCathodeRearClamp.monitoring.goToWorkPos,
                           enableManualCmds := #statEnableManualCmds,
                           interlockWorkPos := "Unit1.Em6.ControlNodes".cm.Interlock.mendrelCathodeRearClamp.work,
                           interlockHomePos := "Unit1.Em6.ControlNodes".cm.Interlock.mendrelCathodeRearClamp.home,
                           configuration := "Unit1.Em6.Config".cmMendrelCathodeRearClamp,
                           moduleInterface := "Unit1.Em6.HmiInterface".cmMendrelCathodeRearClamp,
                           controlNode := "Unit1.Em6.ControlNodes".cmMendrelCathodeRearClamp,
                           goToWorkPos => "BA040AZSPM04.10");
END_REGION

REGION Network 326: CmStackTableVaccum Interlock
   RUNG wire#powerrail
      Coil( "Unit1.Em6.ControlNodes".cm.Interlock.stackTableVaccum.home )
   END_RUNG
   RUNG wire#powerrail
      Coil( "Unit1.Em6.ControlNodes".cm.Interlock.stackTableVaccum.work )
   END_RUNG
   // the same network as SCL:
   "Unit1.Em6.ControlNodes".cm.Interlock.stackTableVaccum.home := TRUE;
   "Unit1.Em6.ControlNodes".cm.Interlock.stackTableVaccum.work := TRUE;
END_REGION

REGION Network 327: CmStackTableVaccum Commands
   RUNG wire#powerrail
      I_Contact( "Unit1.Em6.ControlNodes".gaugeRnR."step".action1[410] )
      Not()
      Coil( "Unit1.Em6.ControlNodes".cmStackTableVaccum.commands.commandHomePos )
   END_RUNG
   RUNG wire#powerrail
      I_Contact( "Unit1.Em6.ControlNodes".gaugeRnR."step".action1[210] )
      Not()
      Coil( "Unit1.Em6.ControlNodes".cmStackTableVaccum.commands.commandWorkPos )
   END_RUNG
   // the same network as SCL:
   "Unit1.Em6.ControlNodes".cmStackTableVaccum.commands.commandHomePos := NOT (NOT "Unit1.Em6.ControlNodes".gaugeRnR."step".action1[410]);
   "Unit1.Em6.ControlNodes".cmStackTableVaccum.commands.commandWorkPos := NOT (NOT "Unit1.Em6.ControlNodes".gaugeRnR."step".action1[210]);
END_REGION

REGION Network 328: Call instCmStackTableVaccum
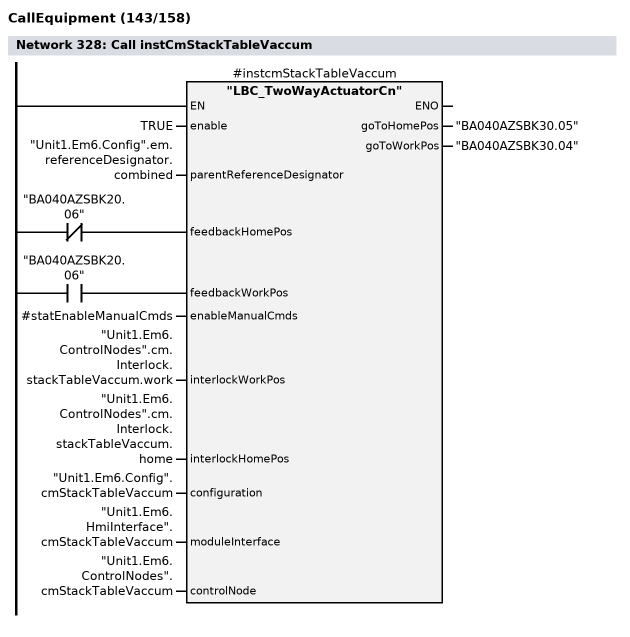
   RUNG wire#powerrail
      #instcmStackTableVaccum(feedbackHomePos := wire#w1, feedbackWorkPos := wire#w2, enable := TRUE, parentReferenceDesignator := "Unit1.Em6.Config".em.referenceDesignator.combined, enableManualCmds := #statEnableManualCmds, interlockWorkPos := "Unit1.Em6.ControlNodes".cm.Interlock.stackTableVaccum.work, interlockHomePos := "Unit1.Em6.ControlNodes".cm.Interlock.stackTableVaccum.home, configuration := "Unit1.Em6.Config".cmStackTableVaccum, moduleInterface := "Unit1.Em6.HmiInterface".cmStackTableVaccum, controlNode := "Unit1.Em6.ControlNodes".cmStackTableVaccum, goToHomePos => "BA040AZSBK30.05", goToWorkPos => "BA040AZSBK30.04")
   END_RUNG
   RUNG wire#powerrail
      I_Contact( "BA040AZSBK20.06" )
   END_RUNG wire#w1
   RUNG wire#powerrail
      Contact( "BA040AZSBK20.06" )
   END_RUNG wire#w2
   // the same network as SCL:
   #instcmStackTableVaccum(enable := TRUE,   // "LBC_TwoWayActuatorCn"
                           parentReferenceDesignator := "Unit1.Em6.Config".em.referenceDesignator.combined,
                           feedbackHomePos := NOT "BA040AZSBK20.06",
                           feedbackWorkPos := "BA040AZSBK20.06",
                           enableManualCmds := #statEnableManualCmds,
                           interlockWorkPos := "Unit1.Em6.ControlNodes".cm.Interlock.stackTableVaccum.work,
                           interlockHomePos := "Unit1.Em6.ControlNodes".cm.Interlock.stackTableVaccum.home,
                           configuration := "Unit1.Em6.Config".cmStackTableVaccum,
                           moduleInterface := "Unit1.Em6.HmiInterface".cmStackTableVaccum,
                           controlNode := "Unit1.Em6.ControlNodes".cmStackTableVaccum,
                           goToHomePos => "BA040AZSBK30.05",
                           goToWorkPos => "BA040AZSBK30.04");
END_REGION

REGION Network 330: CmStackTableGapPadUpDown Interlock
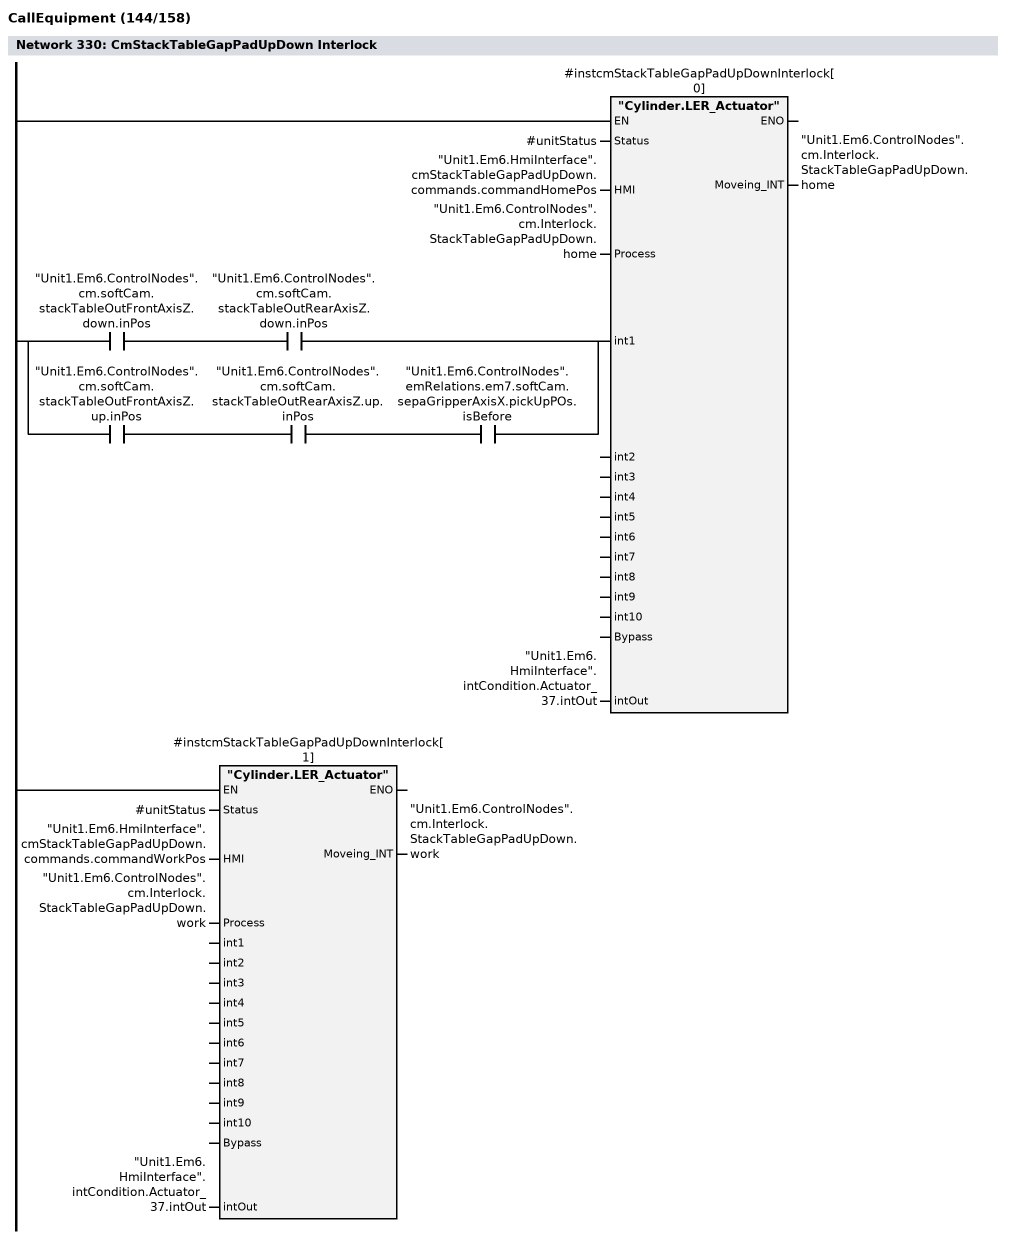
   RUNG wire#powerrail
      #instcmStackTableGapPadUpDownInterlock[0](int1 := wire#w1, Status := #unitStatus, HMI := "Unit1.Em6.HmiInterface".cmStackTableGapPadUpDown.commands.commandHomePos, Process := "Unit1.Em6.ControlNodes".cm.Interlock.StackTableGapPadUpDown.home, int2 :=, int3 :=, int4 :=, int5 :=, int6 :=, int7 :=, int8 :=, int9 :=, int10 :=, Bypass :=, intOut := "Unit1.Em6.HmiInterface".intCondition.Actuator_37.intOut, Moveing_INT => "Unit1.Em6.ControlNodes".cm.Interlock.StackTableGapPadUpDown.home)
   END_RUNG
   RUNG wire#powerrail
      Contact( "Unit1.Em6.ControlNodes".cm.softCam.stackTableOutFrontAxisZ.down.inPos )
      Contact( "Unit1.Em6.ControlNodes".cm.softCam.stackTableOutRearAxisZ.down.inPos )
   END_RUNG wire#w1
   RUNG wire#powerrail
      Contact( "Unit1.Em6.ControlNodes".cm.softCam.stackTableOutFrontAxisZ.up.inPos )
      Contact( "Unit1.Em6.ControlNodes".cm.softCam.stackTableOutRearAxisZ.up.inPos )
      Contact( "Unit1.Em6.ControlNodes".emRelations.em7.softCam.sepaGripperAxisX.pickUpPOs.isBefore )
   END_RUNG wire#w1
   RUNG wire#powerrail
      #instcmStackTableGapPadUpDownInterlock[1](Status := #unitStatus, HMI := "Unit1.Em6.HmiInterface".cmStackTableGapPadUpDown.commands.commandWorkPos, Process := "Unit1.Em6.ControlNodes".cm.Interlock.StackTableGapPadUpDown.work, int1 :=, int2 :=, int3 :=, int4 :=, int5 :=, int6 :=, int7 :=, int8 :=, int9 :=, int10 :=, Bypass :=, intOut := "Unit1.Em6.HmiInterface".intCondition.Actuator_37.intOut, Moveing_INT => "Unit1.Em6.ControlNodes".cm.Interlock.StackTableGapPadUpDown.work)
   END_RUNG
   // the same network as SCL:
   #instcmStackTableGapPadUpDownInterlock[0](Status := #unitStatus,   // "Cylinder.LER_Actuator"
                           HMI := "Unit1.Em6.HmiInterface".cmStackTableGapPadUpDown.commands.commandHomePos,
                           Process := "Unit1.Em6.ControlNodes".cm.Interlock.StackTableGapPadUpDown.home,
                           int1 := ("Unit1.Em6.ControlNodes".cm.softCam.stackTableOutFrontAxisZ.down.inPos AND "Unit1.Em6.ControlNodes".cm.softCam.stackTableOutRearAxisZ.down.inPos) OR ("Unit1.Em6.ControlNodes".cm.softCam.stackTableOutFrontAxisZ.up.inPos AND "Unit1.Em6.ControlNodes".cm.softCam.stackTableOutRearAxisZ.up.inPos AND "Unit1.Em6.ControlNodes".emRelations.em7.softCam.sepaGripperAxisX.pickUpPOs.isBefore),
                           intOut := "Unit1.Em6.HmiInterface".intCondition.Actuator_37.intOut,
                           Moveing_INT => "Unit1.Em6.ControlNodes".cm.Interlock.StackTableGapPadUpDown.home);
   #instcmStackTableGapPadUpDownInterlock[1](Status := #unitStatus,   // "Cylinder.LER_Actuator"
                           HMI := "Unit1.Em6.HmiInterface".cmStackTableGapPadUpDown.commands.commandWorkPos,
                           Process := "Unit1.Em6.ControlNodes".cm.Interlock.StackTableGapPadUpDown.work,
                           intOut := "Unit1.Em6.HmiInterface".intCondition.Actuator_37.intOut,
                           Moveing_INT => "Unit1.Em6.ControlNodes".cm.Interlock.StackTableGapPadUpDown.work);
END_REGION

REGION Network 331: CmStackTableGapPadUpDown Commands
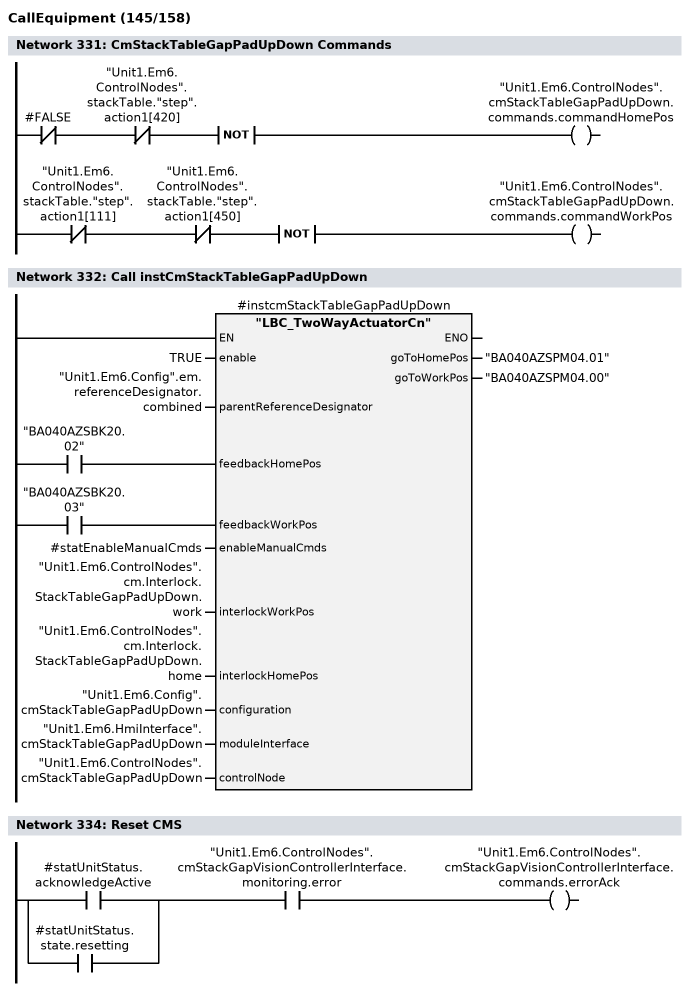
   RUNG wire#powerrail
      I_Contact( #FALSE )
      I_Contact( "Unit1.Em6.ControlNodes".stackTable."step".action1[420] )
      Not()
      Coil( "Unit1.Em6.ControlNodes".cmStackTableGapPadUpDown.commands.commandHomePos )
   END_RUNG
   RUNG wire#powerrail
      I_Contact( "Unit1.Em6.ControlNodes".stackTable."step".action1[111] )
      I_Contact( "Unit1.Em6.ControlNodes".stackTable."step".action1[450] )
      Not()
      Coil( "Unit1.Em6.ControlNodes".cmStackTableGapPadUpDown.commands.commandWorkPos )
   END_RUNG
   // the same network as SCL:
   "Unit1.Em6.ControlNodes".cmStackTableGapPadUpDown.commands.commandHomePos := NOT (NOT #FALSE AND NOT "Unit1.Em6.ControlNodes".stackTable."step".action1[420]);
   "Unit1.Em6.ControlNodes".cmStackTableGapPadUpDown.commands.commandWorkPos := NOT (NOT "Unit1.Em6.ControlNodes".stackTable."step".action1[111] AND NOT "Unit1.Em6.ControlNodes".stackTable."step".action1[450]);
END_REGION

REGION Network 332: Call instCmStackTableGapPadUpDown
   RUNG wire#powerrail
      #instcmStackTableGapPadUpDown(feedbackHomePos := wire#w1, feedbackWorkPos := wire#w2, enable := TRUE, parentReferenceDesignator := "Unit1.Em6.Config".em.referenceDesignator.combined, enableManualCmds := #statEnableManualCmds, interlockWorkPos := "Unit1.Em6.ControlNodes".cm.Interlock.StackTableGapPadUpDown.work, interlockHomePos := "Unit1.Em6.ControlNodes".cm.Interlock.StackTableGapPadUpDown.home, configuration := "Unit1.Em6.Config".cmStackTableGapPadUpDown, moduleInterface := "Unit1.Em6.HmiInterface".cmStackTableGapPadUpDown, controlNode := "Unit1.Em6.ControlNodes".cmStackTableGapPadUpDown, goToHomePos => "BA040AZSPM04.01", goToWorkPos => "BA040AZSPM04.00")
   END_RUNG
   RUNG wire#powerrail
      Contact( "BA040AZSBK20.02" )
   END_RUNG wire#w1
   RUNG wire#powerrail
      Contact( "BA040AZSBK20.03" )
   END_RUNG wire#w2
   // the same network as SCL:
   #instcmStackTableGapPadUpDown(enable := TRUE,   // "LBC_TwoWayActuatorCn"
                           parentReferenceDesignator := "Unit1.Em6.Config".em.referenceDesignator.combined,
                           feedbackHomePos := "BA040AZSBK20.02",
                           feedbackWorkPos := "BA040AZSBK20.03",
                           enableManualCmds := #statEnableManualCmds,
                           interlockWorkPos := "Unit1.Em6.ControlNodes".cm.Interlock.StackTableGapPadUpDown.work,
                           interlockHomePos := "Unit1.Em6.ControlNodes".cm.Interlock.StackTableGapPadUpDown.home,
                           configuration := "Unit1.Em6.Config".cmStackTableGapPadUpDown,
                           moduleInterface := "Unit1.Em6.HmiInterface".cmStackTableGapPadUpDown,
                           controlNode := "Unit1.Em6.ControlNodes".cmStackTableGapPadUpDown,
                           goToHomePos => "BA040AZSPM04.01",
                           goToWorkPos => "BA040AZSPM04.00");
END_REGION

REGION Network 333: ******************** Control Modules (Accessories) ********************
END_REGION

REGION Network 334: Reset CMS
   RUNG wire#powerrail
      Contact( #statUnitStatus.acknowledgeActive )
      wire#w1
      Contact( "Unit1.Em6.ControlNodes".cmStackGapVisionControllerInterface.monitoring.error )
      Coil( "Unit1.Em6.ControlNodes".cmStackGapVisionControllerInterface.commands.errorAck )
   END_RUNG
   RUNG wire#powerrail
      Contact( #statUnitStatus.state.resetting )
   END_RUNG wire#w1
   // the same network as SCL:
   "Unit1.Em6.ControlNodes".cmStackGapVisionControllerInterface.commands.errorAck := (#statUnitStatus.acknowledgeActive OR #statUnitStatus.state.resetting) AND "Unit1.Em6.ControlNodes".cmStackGapVisionControllerInterface.monitoring.error;
END_REGION

REGION Network 335: CmGapVisionControllerInterface Commands
